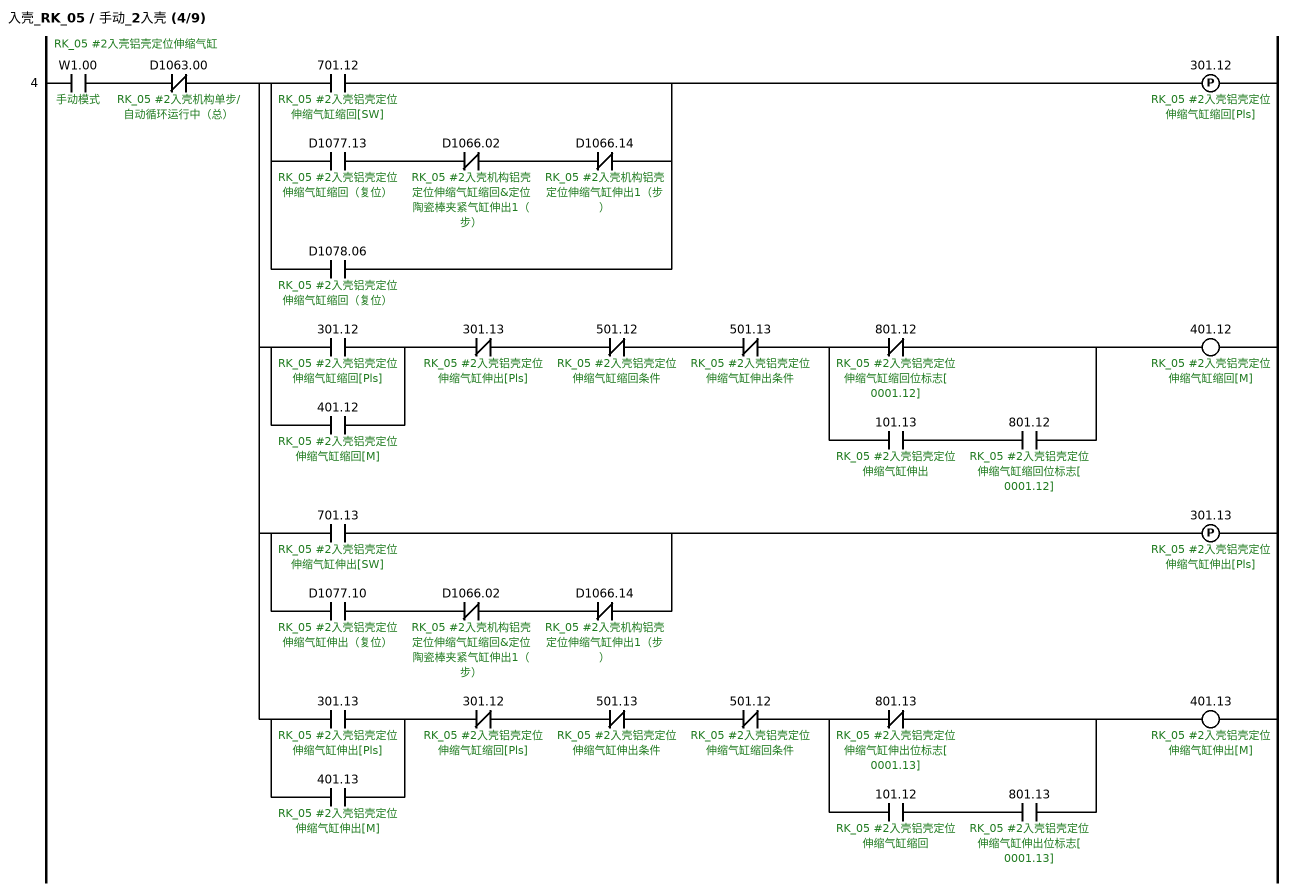
; [picture p432: 入壳_RK_05 / 手动_2入壳, rungs 4-4]
; rung 4: RK_05 #2入壳铝壳定位伸缩气缸
LD W1.00  ; 手动模式
ANDNOT D1063.00  ; RK_05 #2入壳机构单步/自动循环运行中（总）
OUT TR0
LD 701.12  ; RK_05 #2入壳铝壳定位伸缩气缸缩回[SW]
LD D1077.13  ; RK_05 #2入壳铝壳定位伸缩气缸缩回（复位）
ANDNOT D1066.02  ; RK_05 #2入壳机构铝壳定位伸缩气缸缩回&定位陶瓷棒夹紧气缸伸出1（步）
ANDNOT D1066.14  ; RK_05 #2入壳机构铝壳定位伸缩气缸伸出1（步）
ORLD
OR D1078.06  ; RK_05 #2入壳铝壳定位伸缩气缸缩回（复位）
ANDLD
DIFU(013) 301.12  ; RK_05 #2入壳铝壳定位伸缩气缸缩回[Pls]
LD TR0
LD 301.12  ; RK_05 #2入壳铝壳定位伸缩气缸缩回[Pls]
OR 401.12  ; RK_05 #2入壳铝壳定位伸缩气缸缩回[M]
ANDLD
ANDNOT 301.13  ; RK_05 #2入壳铝壳定位伸缩气缸伸出[Pls]
ANDNOT 501.12  ; RK_05 #2入壳铝壳定位伸缩气缸缩回条件
ANDNOT 501.13  ; RK_05 #2入壳铝壳定位伸缩气缸伸出条件
LDNOT 801.12  ; RK_05 #2入壳铝壳定位伸缩气缸缩回位标志[0001.12]
LD 101.13  ; RK_05 #2入壳铝壳定位伸缩气缸伸出
AND 801.12  ; RK_05 #2入壳铝壳定位伸缩气缸缩回位标志[0001.12]
ORLD
ANDLD
OUT 401.12  ; RK_05 #2入壳铝壳定位伸缩气缸缩回[M]
LD TR0
LD 701.13  ; RK_05 #2入壳铝壳定位伸缩气缸伸出[SW]
LD D1077.10  ; RK_05 #2入壳铝壳定位伸缩气缸伸出（复位）
ANDNOT D1066.02  ; RK_05 #2入壳机构铝壳定位伸缩气缸缩回&定位陶瓷棒夹紧气缸伸出1（步）
ANDNOT D1066.14  ; RK_05 #2入壳机构铝壳定位伸缩气缸伸出1（步）
ORLD
ANDLD
DIFU(013) 301.13  ; RK_05 #2入壳铝壳定位伸缩气缸伸出[Pls]
LD TR0
LD 301.13  ; RK_05 #2入壳铝壳定位伸缩气缸伸出[Pls]
OR 401.13  ; RK_05 #2入壳铝壳定位伸缩气缸伸出[M]
ANDLD
ANDNOT 301.12  ; RK_05 #2入壳铝壳定位伸缩气缸缩回[Pls]
ANDNOT 501.13  ; RK_05 #2入壳铝壳定位伸缩气缸伸出条件
ANDNOT 501.12  ; RK_05 #2入壳铝壳定位伸缩气缸缩回条件
LDNOT 801.13  ; RK_05 #2入壳铝壳定位伸缩气缸伸出位标志[0001.13]
LD 101.12  ; RK_05 #2入壳铝壳定位伸缩气缸缩回
AND 801.13  ; RK_05 #2入壳铝壳定位伸缩气缸伸出位标志[0001.13]
ORLD
ANDLD
OUT 401.13  ; RK_05 #2入壳铝壳定位伸缩气缸伸出[M]

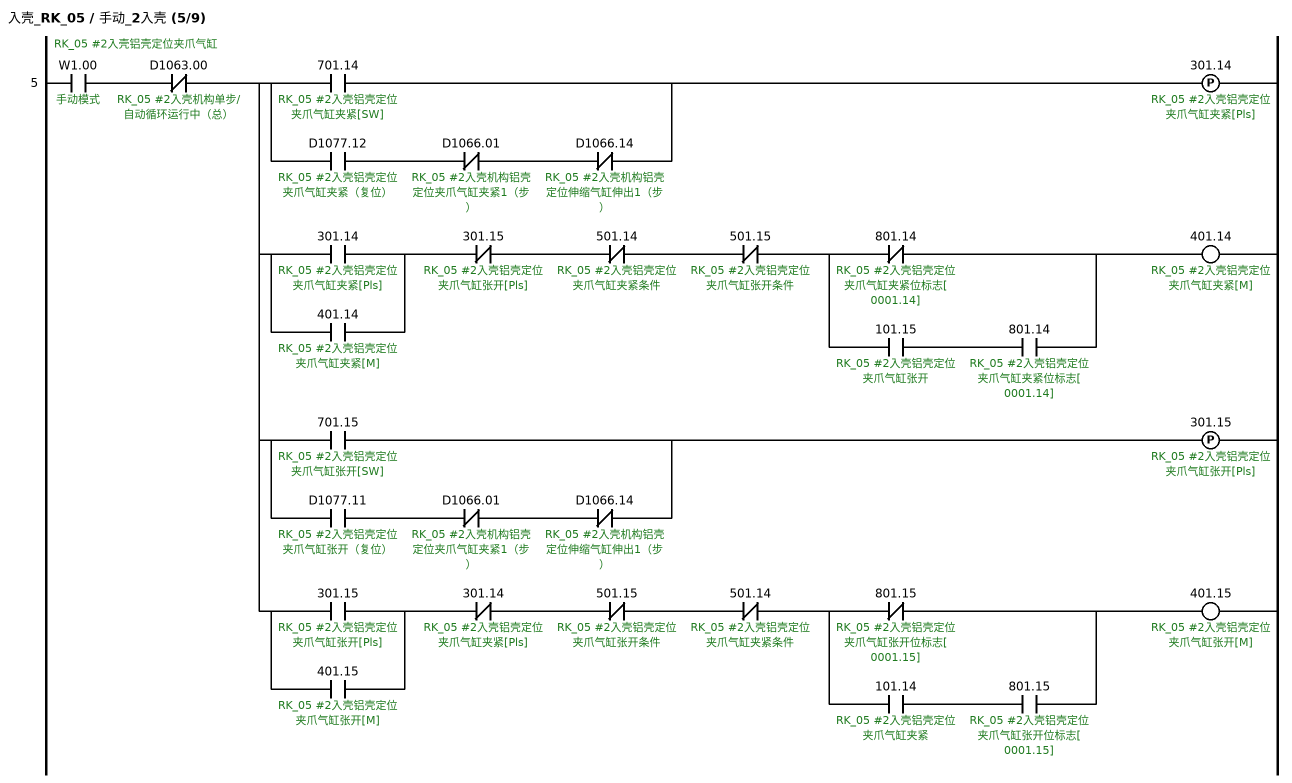
; rung 5: RK_05 #2入壳铝壳定位夹爪气缸
LD W1.00  ; 手动模式
ANDNOT D1063.00  ; RK_05 #2入壳机构单步/自动循环运行中（总）
OUT TR0
LD 701.14  ; RK_05 #2入壳铝壳定位夹爪气缸夹紧[SW]
LD D1077.12  ; RK_05 #2入壳铝壳定位夹爪气缸夹紧（复位）
ANDNOT D1066.01  ; RK_05 #2入壳机构铝壳定位夹爪气缸夹紧1（步）
ANDNOT D1066.14  ; RK_05 #2入壳机构铝壳定位伸缩气缸伸出1（步）
ORLD
ANDLD
DIFU(013) 301.14  ; RK_05 #2入壳铝壳定位夹爪气缸夹紧[Pls]
LD TR0
LD 301.14  ; RK_05 #2入壳铝壳定位夹爪气缸夹紧[Pls]
OR 401.14  ; RK_05 #2入壳铝壳定位夹爪气缸夹紧[M]
ANDLD
ANDNOT 301.15  ; RK_05 #2入壳铝壳定位夹爪气缸张开[Pls]
ANDNOT 501.14  ; RK_05 #2入壳铝壳定位夹爪气缸夹紧条件
ANDNOT 501.15  ; RK_05 #2入壳铝壳定位夹爪气缸张开条件
LDNOT 801.14  ; RK_05 #2入壳铝壳定位夹爪气缸夹紧位标志[0001.14]
LD 101.15  ; RK_05 #2入壳铝壳定位夹爪气缸张开
AND 801.14  ; RK_05 #2入壳铝壳定位夹爪气缸夹紧位标志[0001.14]
ORLD
ANDLD
OUT 401.14  ; RK_05 #2入壳铝壳定位夹爪气缸夹紧[M]
LD TR0
LD 701.15  ; RK_05 #2入壳铝壳定位夹爪气缸张开[SW]
LD D1077.11  ; RK_05 #2入壳铝壳定位夹爪气缸张开（复位）
ANDNOT D1066.01  ; RK_05 #2入壳机构铝壳定位夹爪气缸夹紧1（步）
ANDNOT D1066.14  ; RK_05 #2入壳机构铝壳定位伸缩气缸伸出1（步）
ORLD
ANDLD
DIFU(013) 301.15  ; RK_05 #2入壳铝壳定位夹爪气缸张开[Pls]
LD TR0
LD 301.15  ; RK_05 #2入壳铝壳定位夹爪气缸张开[Pls]
OR 401.15  ; RK_05 #2入壳铝壳定位夹爪气缸张开[M]
ANDLD
ANDNOT 301.14  ; RK_05 #2入壳铝壳定位夹爪气缸夹紧[Pls]
ANDNOT 501.15  ; RK_05 #2入壳铝壳定位夹爪气缸张开条件
ANDNOT 501.14  ; RK_05 #2入壳铝壳定位夹爪气缸夹紧条件
LDNOT 801.15  ; RK_05 #2入壳铝壳定位夹爪气缸张开位标志[0001.15]
LD 101.14  ; RK_05 #2入壳铝壳定位夹爪气缸夹紧
AND 801.15  ; RK_05 #2入壳铝壳定位夹爪气缸张开位标志[0001.15]
ORLD
ANDLD
OUT 401.15  ; RK_05 #2入壳铝壳定位夹爪气缸张开[M]

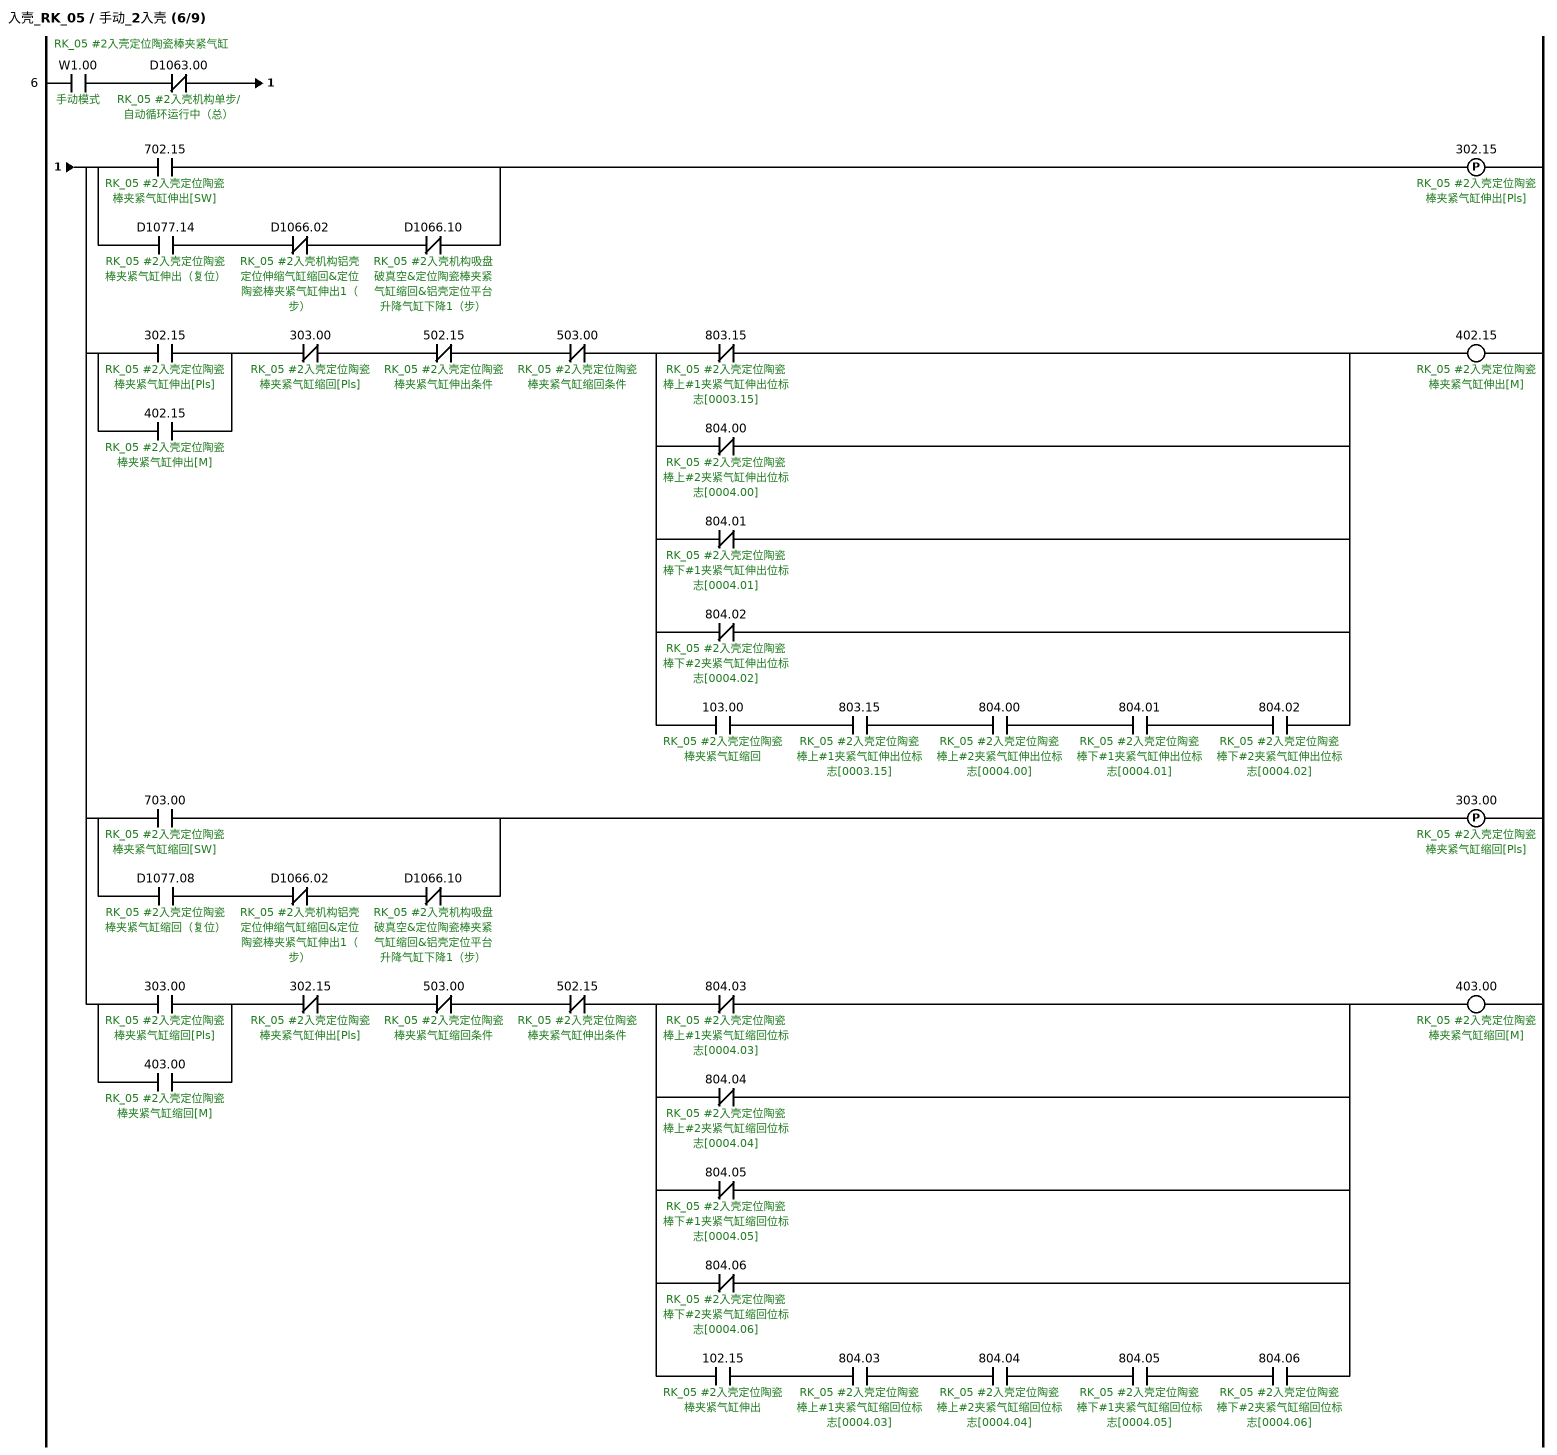
; rung 6: RK_05 #2入壳定位陶瓷棒夹紧气缸
LD W1.00  ; 手动模式
ANDNOT D1063.00  ; RK_05 #2入壳机构单步/自动循环运行中（总）
OUT TR0
LD 702.15  ; RK_05 #2入壳定位陶瓷棒夹紧气缸伸出[SW]
LD D1077.14  ; RK_05 #2入壳定位陶瓷棒夹紧气缸伸出（复位）
ANDNOT D1066.02  ; RK_05 #2入壳机构铝壳定位伸缩气缸缩回&定位陶瓷棒夹紧气缸伸出1（步）
ANDNOT D1066.10  ; RK_05 #2入壳机构吸盘破真空&定位陶瓷棒夹紧气缸缩回&铝壳定位平台升降气缸下降1（步）
ORLD
ANDLD
DIFU(013) 302.15  ; RK_05 #2入壳定位陶瓷棒夹紧气缸伸出[Pls]
LD TR0
LD 302.15  ; RK_05 #2入壳定位陶瓷棒夹紧气缸伸出[Pls]
OR 402.15  ; RK_05 #2入壳定位陶瓷棒夹紧气缸伸出[M]
ANDLD
ANDNOT 303.00  ; RK_05 #2入壳定位陶瓷棒夹紧气缸缩回[Pls]
ANDNOT 502.15  ; RK_05 #2入壳定位陶瓷棒夹紧气缸伸出条件
ANDNOT 503.00  ; RK_05 #2入壳定位陶瓷棒夹紧气缸缩回条件
LDNOT 803.15  ; RK_05 #2入壳定位陶瓷棒上#1夹紧气缸伸出位标志[0003.15]
ORNOT 804.00  ; RK_05 #2入壳定位陶瓷棒上#2夹紧气缸伸出位标志[0004.00]
ORNOT 804.01  ; RK_05 #2入壳定位陶瓷棒下#1夹紧气缸伸出位标志[0004.01]
ORNOT 804.02  ; RK_05 #2入壳定位陶瓷棒下#2夹紧气缸伸出位标志[0004.02]
LD 103.00  ; RK_05 #2入壳定位陶瓷棒夹紧气缸缩回
AND 803.15  ; RK_05 #2入壳定位陶瓷棒上#1夹紧气缸伸出位标志[0003.15]
AND 804.00  ; RK_05 #2入壳定位陶瓷棒上#2夹紧气缸伸出位标志[0004.00]
AND 804.01  ; RK_05 #2入壳定位陶瓷棒下#1夹紧气缸伸出位标志[0004.01]
AND 804.02  ; RK_05 #2入壳定位陶瓷棒下#2夹紧气缸伸出位标志[0004.02]
ORLD
ANDLD
OUT 402.15  ; RK_05 #2入壳定位陶瓷棒夹紧气缸伸出[M]
LD TR0
LD 703.00  ; RK_05 #2入壳定位陶瓷棒夹紧气缸缩回[SW]
LD D1077.08  ; RK_05 #2入壳定位陶瓷棒夹紧气缸缩回（复位）
ANDNOT D1066.02  ; RK_05 #2入壳机构铝壳定位伸缩气缸缩回&定位陶瓷棒夹紧气缸伸出1（步）
ANDNOT D1066.10  ; RK_05 #2入壳机构吸盘破真空&定位陶瓷棒夹紧气缸缩回&铝壳定位平台升降气缸下降1（步）
ORLD
ANDLD
DIFU(013) 303.00  ; RK_05 #2入壳定位陶瓷棒夹紧气缸缩回[Pls]
LD TR0
LD 303.00  ; RK_05 #2入壳定位陶瓷棒夹紧气缸缩回[Pls]
OR 403.00  ; RK_05 #2入壳定位陶瓷棒夹紧气缸缩回[M]
ANDLD
ANDNOT 302.15  ; RK_05 #2入壳定位陶瓷棒夹紧气缸伸出[Pls]
ANDNOT 503.00  ; RK_05 #2入壳定位陶瓷棒夹紧气缸缩回条件
ANDNOT 502.15  ; RK_05 #2入壳定位陶瓷棒夹紧气缸伸出条件
LDNOT 804.03  ; RK_05 #2入壳定位陶瓷棒上#1夹紧气缸缩回位标志[0004.03]
ORNOT 804.04  ; RK_05 #2入壳定位陶瓷棒上#2夹紧气缸缩回位标志[0004.04]
ORNOT 804.05  ; RK_05 #2入壳定位陶瓷棒下#1夹紧气缸缩回位标志[0004.05]
ORNOT 804.06  ; RK_05 #2入壳定位陶瓷棒下#2夹紧气缸缩回位标志[0004.06]
LD 102.15  ; RK_05 #2入壳定位陶瓷棒夹紧气缸伸出
AND 804.03  ; RK_05 #2入壳定位陶瓷棒上#1夹紧气缸缩回位标志[0004.03]
AND 804.04  ; RK_05 #2入壳定位陶瓷棒上#2夹紧气缸缩回位标志[0004.04]
AND 804.05  ; RK_05 #2入壳定位陶瓷棒下#1夹紧气缸缩回位标志[0004.05]
AND 804.06  ; RK_05 #2入壳定位陶瓷棒下#2夹紧气缸缩回位标志[0004.06]
ORLD
ANDLD
OUT 403.00  ; RK_05 #2入壳定位陶瓷棒夹紧气缸缩回[M]

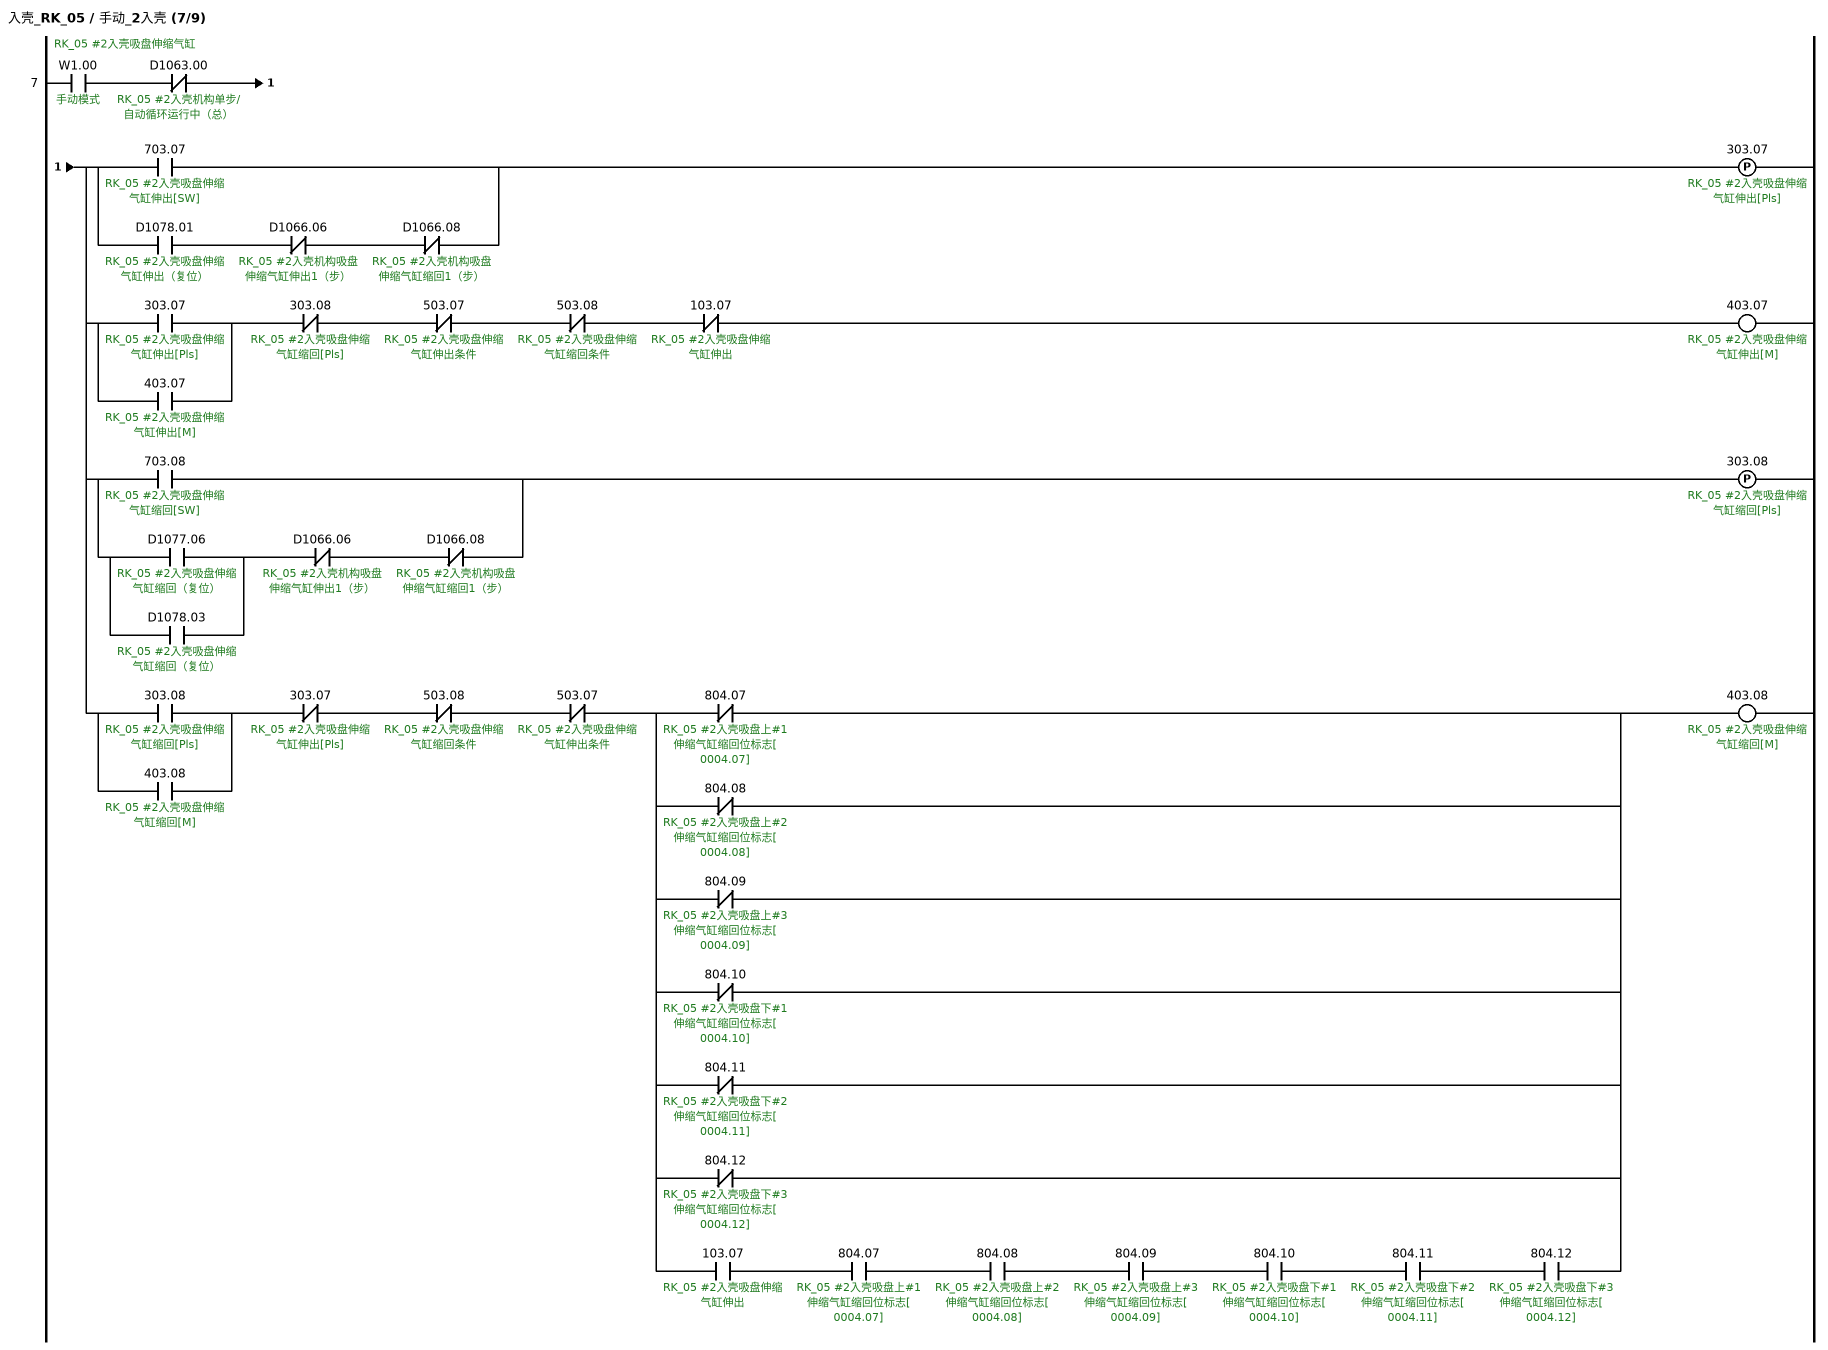
; rung 7: RK_05 #2入壳吸盘伸缩气缸
LD W1.00  ; 手动模式
ANDNOT D1063.00  ; RK_05 #2入壳机构单步/自动循环运行中（总）
OUT TR0
LD 703.07  ; RK_05 #2入壳吸盘伸缩气缸伸出[SW]
LD D1078.01  ; RK_05 #2入壳吸盘伸缩气缸伸出（复位）
ANDNOT D1066.06  ; RK_05 #2入壳机构吸盘伸缩气缸伸出1（步）
ANDNOT D1066.08  ; RK_05 #2入壳机构吸盘伸缩气缸缩回1（步）
ORLD
ANDLD
DIFU(013) 303.07  ; RK_05 #2入壳吸盘伸缩气缸伸出[Pls]
LD TR0
LD 303.07  ; RK_05 #2入壳吸盘伸缩气缸伸出[Pls]
OR 403.07  ; RK_05 #2入壳吸盘伸缩气缸伸出[M]
ANDLD
ANDNOT 303.08  ; RK_05 #2入壳吸盘伸缩气缸缩回[Pls]
ANDNOT 503.07  ; RK_05 #2入壳吸盘伸缩气缸伸出条件
ANDNOT 503.08  ; RK_05 #2入壳吸盘伸缩气缸缩回条件
ANDNOT 103.07  ; RK_05 #2入壳吸盘伸缩气缸伸出
OUT 403.07  ; RK_05 #2入壳吸盘伸缩气缸伸出[M]
LD TR0
LD 703.08  ; RK_05 #2入壳吸盘伸缩气缸缩回[SW]
LD D1077.06  ; RK_05 #2入壳吸盘伸缩气缸缩回（复位）
OR D1078.03  ; RK_05 #2入壳吸盘伸缩气缸缩回（复位）
ANDNOT D1066.06  ; RK_05 #2入壳机构吸盘伸缩气缸伸出1（步）
ANDNOT D1066.08  ; RK_05 #2入壳机构吸盘伸缩气缸缩回1（步）
ORLD
ANDLD
DIFU(013) 303.08  ; RK_05 #2入壳吸盘伸缩气缸缩回[Pls]
LD TR0
LD 303.08  ; RK_05 #2入壳吸盘伸缩气缸缩回[Pls]
OR 403.08  ; RK_05 #2入壳吸盘伸缩气缸缩回[M]
ANDLD
ANDNOT 303.07  ; RK_05 #2入壳吸盘伸缩气缸伸出[Pls]
ANDNOT 503.08  ; RK_05 #2入壳吸盘伸缩气缸缩回条件
ANDNOT 503.07  ; RK_05 #2入壳吸盘伸缩气缸伸出条件
LDNOT 804.07  ; RK_05 #2入壳吸盘上#1伸缩气缸缩回位标志[0004.07]
ORNOT 804.08  ; RK_05 #2入壳吸盘上#2伸缩气缸缩回位标志[0004.08]
ORNOT 804.09  ; RK_05 #2入壳吸盘上#3伸缩气缸缩回位标志[0004.09]
ORNOT 804.10  ; RK_05 #2入壳吸盘下#1伸缩气缸缩回位标志[0004.10]
ORNOT 804.11  ; RK_05 #2入壳吸盘下#2伸缩气缸缩回位标志[0004.11]
ORNOT 804.12  ; RK_05 #2入壳吸盘下#3伸缩气缸缩回位标志[0004.12]
LD 103.07  ; RK_05 #2入壳吸盘伸缩气缸伸出
AND 804.07  ; RK_05 #2入壳吸盘上#1伸缩气缸缩回位标志[0004.07]
AND 804.08  ; RK_05 #2入壳吸盘上#2伸缩气缸缩回位标志[0004.08]
AND 804.09  ; RK_05 #2入壳吸盘上#3伸缩气缸缩回位标志[0004.09]
AND 804.10  ; RK_05 #2入壳吸盘下#1伸缩气缸缩回位标志[0004.10]
AND 804.11  ; RK_05 #2入壳吸盘下#2伸缩气缸缩回位标志[0004.11]
AND 804.12  ; RK_05 #2入壳吸盘下#3伸缩气缸缩回位标志[0004.12]
ORLD
ANDLD
OUT 403.08  ; RK_05 #2入壳吸盘伸缩气缸缩回[M]

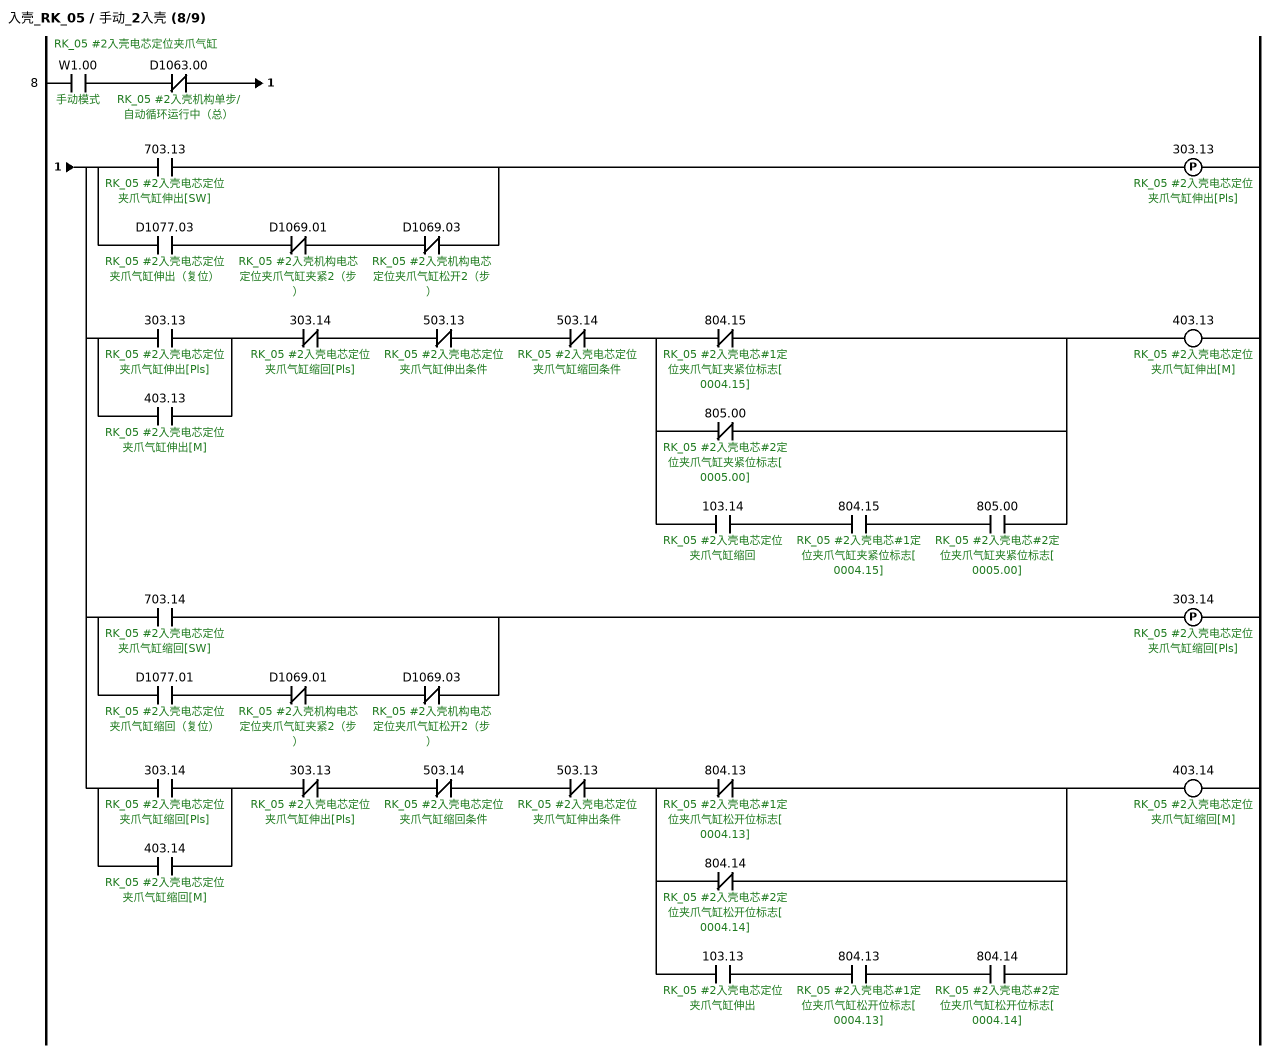
; rung 8: RK_05 #2入壳电芯定位夹爪气缸
LD W1.00  ; 手动模式
ANDNOT D1063.00  ; RK_05 #2入壳机构单步/自动循环运行中（总）
OUT TR0
LD 703.13  ; RK_05 #2入壳电芯定位夹爪气缸伸出[SW]
LD D1077.03  ; RK_05 #2入壳电芯定位夹爪气缸伸出（复位）
ANDNOT D1069.01  ; RK_05 #2入壳机构电芯定位夹爪气缸夹紧2（步）
ANDNOT D1069.03  ; RK_05 #2入壳机构电芯定位夹爪气缸松开2（步）
ORLD
ANDLD
DIFU(013) 303.13  ; RK_05 #2入壳电芯定位夹爪气缸伸出[Pls]
LD TR0
LD 303.13  ; RK_05 #2入壳电芯定位夹爪气缸伸出[Pls]
OR 403.13  ; RK_05 #2入壳电芯定位夹爪气缸伸出[M]
ANDLD
ANDNOT 303.14  ; RK_05 #2入壳电芯定位夹爪气缸缩回[Pls]
ANDNOT 503.13  ; RK_05 #2入壳电芯定位夹爪气缸伸出条件
ANDNOT 503.14  ; RK_05 #2入壳电芯定位夹爪气缸缩回条件
LDNOT 804.15  ; RK_05 #2入壳电芯#1定位夹爪气缸夹紧位标志[0004.15]
ORNOT 805.00  ; RK_05 #2入壳电芯#2定位夹爪气缸夹紧位标志[0005.00]
LD 103.14  ; RK_05 #2入壳电芯定位夹爪气缸缩回
AND 804.15  ; RK_05 #2入壳电芯#1定位夹爪气缸夹紧位标志[0004.15]
AND 805.00  ; RK_05 #2入壳电芯#2定位夹爪气缸夹紧位标志[0005.00]
ORLD
ANDLD
OUT 403.13  ; RK_05 #2入壳电芯定位夹爪气缸伸出[M]
LD TR0
LD 703.14  ; RK_05 #2入壳电芯定位夹爪气缸缩回[SW]
LD D1077.01  ; RK_05 #2入壳电芯定位夹爪气缸缩回（复位）
ANDNOT D1069.01  ; RK_05 #2入壳机构电芯定位夹爪气缸夹紧2（步）
ANDNOT D1069.03  ; RK_05 #2入壳机构电芯定位夹爪气缸松开2（步）
ORLD
ANDLD
DIFU(013) 303.14  ; RK_05 #2入壳电芯定位夹爪气缸缩回[Pls]
LD TR0
LD 303.14  ; RK_05 #2入壳电芯定位夹爪气缸缩回[Pls]
OR 403.14  ; RK_05 #2入壳电芯定位夹爪气缸缩回[M]
ANDLD
ANDNOT 303.13  ; RK_05 #2入壳电芯定位夹爪气缸伸出[Pls]
ANDNOT 503.14  ; RK_05 #2入壳电芯定位夹爪气缸缩回条件
ANDNOT 503.13  ; RK_05 #2入壳电芯定位夹爪气缸伸出条件
LDNOT 804.13  ; RK_05 #2入壳电芯#1定位夹爪气缸松开位标志[0004.13]
ORNOT 804.14  ; RK_05 #2入壳电芯#2定位夹爪气缸松开位标志[0004.14]
LD 103.13  ; RK_05 #2入壳电芯定位夹爪气缸伸出
AND 804.13  ; RK_05 #2入壳电芯#1定位夹爪气缸松开位标志[0004.13]
AND 804.14  ; RK_05 #2入壳电芯#2定位夹爪气缸松开位标志[0004.14]
ORLD
ANDLD
OUT 403.14  ; RK_05 #2入壳电芯定位夹爪气缸缩回[M]

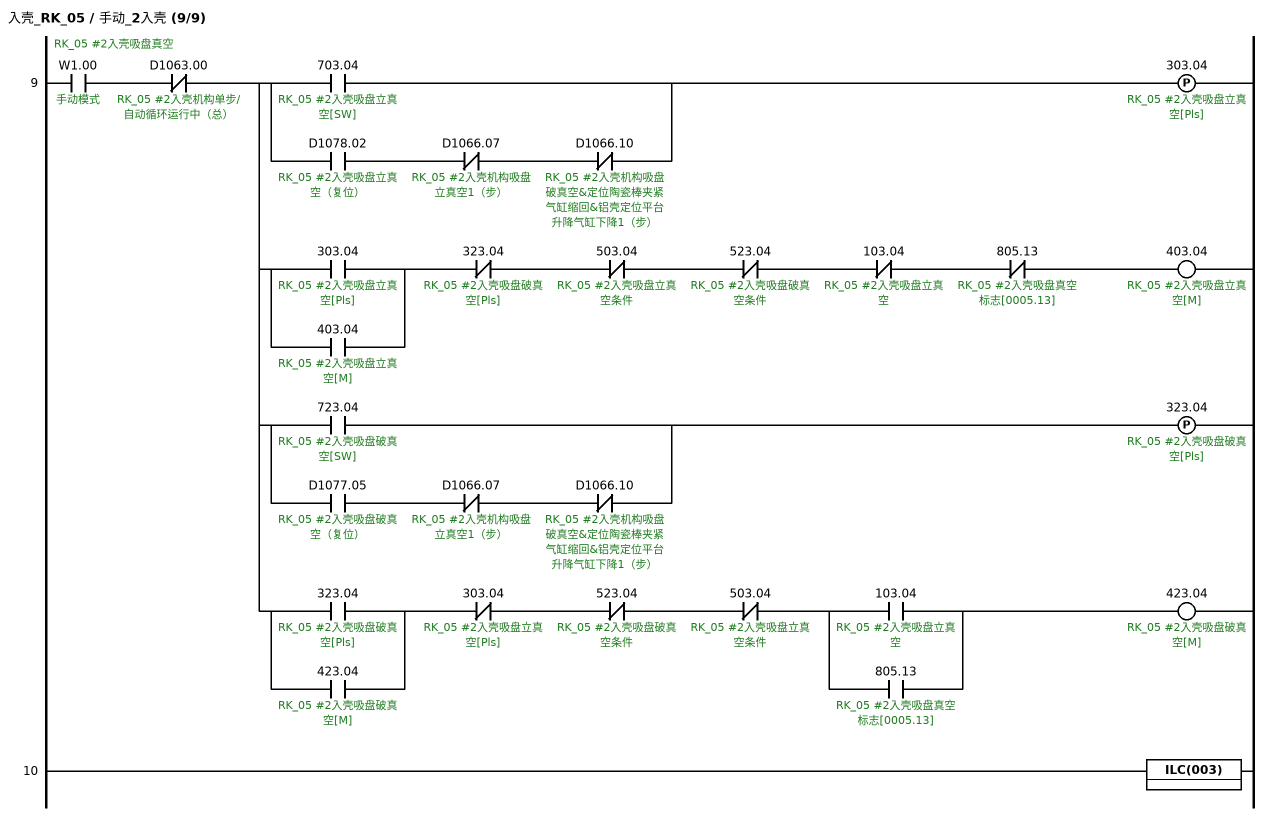
; rung 9: RK_05 #2入壳吸盘真空
LD W1.00  ; 手动模式
ANDNOT D1063.00  ; RK_05 #2入壳机构单步/自动循环运行中（总）
OUT TR0
LD 703.04  ; RK_05 #2入壳吸盘立真空[SW]
LD D1078.02  ; RK_05 #2入壳吸盘立真空（复位）
ANDNOT D1066.07  ; RK_05 #2入壳机构吸盘立真空1（步）
ANDNOT D1066.10  ; RK_05 #2入壳机构吸盘破真空&定位陶瓷棒夹紧气缸缩回&铝壳定位平台升降气缸下降1（步）
ORLD
ANDLD
DIFU(013) 303.04  ; RK_05 #2入壳吸盘立真空[Pls]
LD TR0
LD 303.04  ; RK_05 #2入壳吸盘立真空[Pls]
OR 403.04  ; RK_05 #2入壳吸盘立真空[M]
ANDLD
ANDNOT 323.04  ; RK_05 #2入壳吸盘破真空[Pls]
ANDNOT 503.04  ; RK_05 #2入壳吸盘立真空条件
ANDNOT 523.04  ; RK_05 #2入壳吸盘破真空条件
ANDNOT 103.04  ; RK_05 #2入壳吸盘立真空
ANDNOT 805.13  ; RK_05 #2入壳吸盘真空标志[0005.13]
OUT 403.04  ; RK_05 #2入壳吸盘立真空[M]
LD TR0
LD 723.04  ; RK_05 #2入壳吸盘破真空[SW]
LD D1077.05  ; RK_05 #2入壳吸盘破真空（复位）
ANDNOT D1066.07  ; RK_05 #2入壳机构吸盘立真空1（步）
ANDNOT D1066.10  ; RK_05 #2入壳机构吸盘破真空&定位陶瓷棒夹紧气缸缩回&铝壳定位平台升降气缸下降1（步）
ORLD
ANDLD
DIFU(013) 323.04  ; RK_05 #2入壳吸盘破真空[Pls]
LD TR0
LD 323.04  ; RK_05 #2入壳吸盘破真空[Pls]
OR 423.04  ; RK_05 #2入壳吸盘破真空[M]
ANDLD
ANDNOT 303.04  ; RK_05 #2入壳吸盘立真空[Pls]
ANDNOT 523.04  ; RK_05 #2入壳吸盘破真空条件
ANDNOT 503.04  ; RK_05 #2入壳吸盘立真空条件
LD 103.04  ; RK_05 #2入壳吸盘立真空
OR 805.13  ; RK_05 #2入壳吸盘真空标志[0005.13]
ANDLD
OUT 423.04  ; RK_05 #2入壳吸盘破真空[M]
; rung 10
ILC(003)

### Section 自动_1入壳

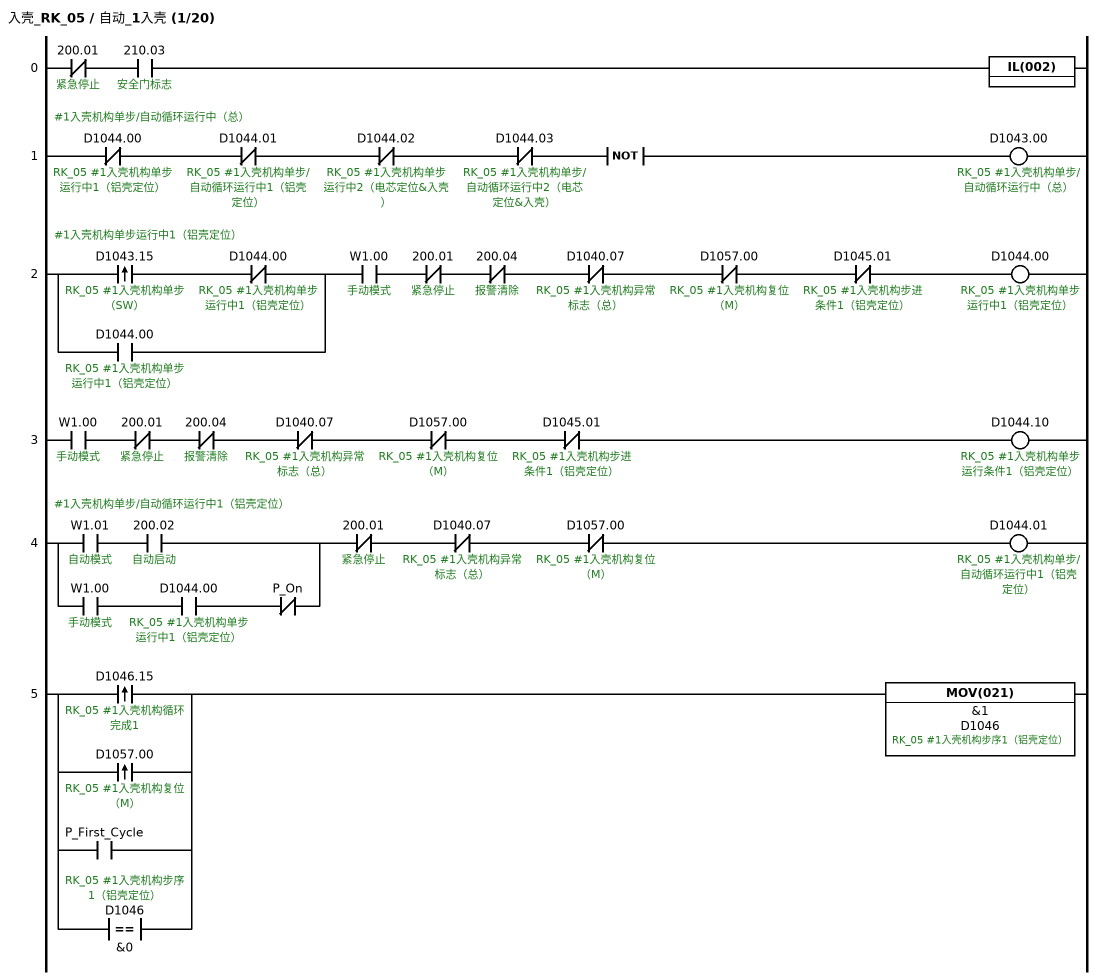
; rung 0
LDNOT 200.01  ; 紧急停止
AND 210.03  ; 安全门标志
IL(002)
; rung 1: #1入壳机构单步/自动循环运行中（总）
LDNOT D1044.00  ; RK_05 #1入壳机构单步运行中1（铝壳定位）
ANDNOT D1044.01  ; RK_05 #1入壳机构单步/自动循环运行中1（铝壳定位）
ANDNOT D1044.02  ; RK_05 #1入壳机构单步运行中2（电芯定位&入壳）
ANDNOT D1044.03  ; RK_05 #1入壳机构单步/自动循环运行中2（电芯定位&入壳）
NOT(520)
OUT D1043.00  ; RK_05 #1入壳机构单步/自动循环运行中（总）
; rung 2: #1入壳机构单步运行中1（铝壳定位）
@LD D1043.15  ; RK_05 #1入壳机构单步（SW）
ANDNOT D1044.00  ; RK_05 #1入壳机构单步运行中1（铝壳定位）
OR D1044.00  ; RK_05 #1入壳机构单步运行中1（铝壳定位）
AND W1.00  ; 手动模式
ANDNOT 200.01  ; 紧急停止
ANDNOT 200.04  ; 报警清除
ANDNOT D1040.07  ; RK_05 #1入壳机构异常标志（总）
ANDNOT D1057.00  ; RK_05 #1入壳机构复位（M）
ANDNOT D1045.01  ; RK_05 #1入壳机构步进条件1（铝壳定位）
OUT D1044.00  ; RK_05 #1入壳机构单步运行中1（铝壳定位）
; rung 3
LD W1.00  ; 手动模式
ANDNOT 200.01  ; 紧急停止
ANDNOT 200.04  ; 报警清除
ANDNOT D1040.07  ; RK_05 #1入壳机构异常标志（总）
ANDNOT D1057.00  ; RK_05 #1入壳机构复位（M）
ANDNOT D1045.01  ; RK_05 #1入壳机构步进条件1（铝壳定位）
OUT D1044.10  ; RK_05 #1入壳机构单步运行条件1（铝壳定位）
; rung 4: #1入壳机构单步/自动循环运行中1（铝壳定位）
LD W1.01  ; 自动模式
AND 200.02  ; 自动启动
LD W1.00  ; 手动模式
AND D1044.00  ; RK_05 #1入壳机构单步运行中1（铝壳定位）
ANDNOT P_On
ORLD
ANDNOT 200.01  ; 紧急停止
ANDNOT D1040.07  ; RK_05 #1入壳机构异常标志（总）
ANDNOT D1057.00  ; RK_05 #1入壳机构复位（M）
OUT D1044.01  ; RK_05 #1入壳机构单步/自动循环运行中1（铝壳定位）
; rung 5
@LD D1046.15  ; RK_05 #1入壳机构循环完成1
@OR D1057.00  ; RK_05 #1入壳机构复位（M）
OR P_First_Cycle
OR=(300) D1046 &0  ; RK_05 #1入壳机构步序1（铝壳定位）
MOV(021) &1 D1046  ; RK_05 #1入壳机构步序1（铝壳定位）

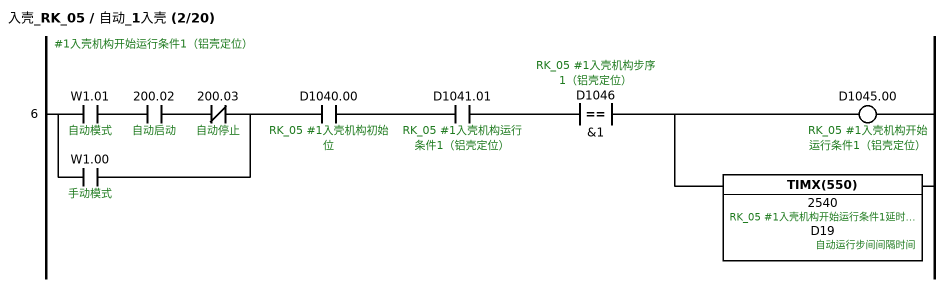
; rung 6: #1入壳机构开始运行条件1（铝壳定位）
LD W1.01  ; 自动模式
AND 200.02  ; 自动启动
ANDNOT 200.03  ; 自动停止
OR W1.00  ; 手动模式
AND D1040.00  ; RK_05 #1入壳机构初始位
AND D1041.01  ; RK_05 #1入壳机构运行条件1（铝壳定位）
AND=(300) D1046 &1  ; RK_05 #1入壳机构步序1（铝壳定位）
OUT D1045.00  ; RK_05 #1入壳机构开始运行条件1（铝壳定位）
TIMX(550) 2540 D19  ; 自动运行步间间隔时间, RK_05 #1入壳机构开始运行条件1延时（铝壳定位）

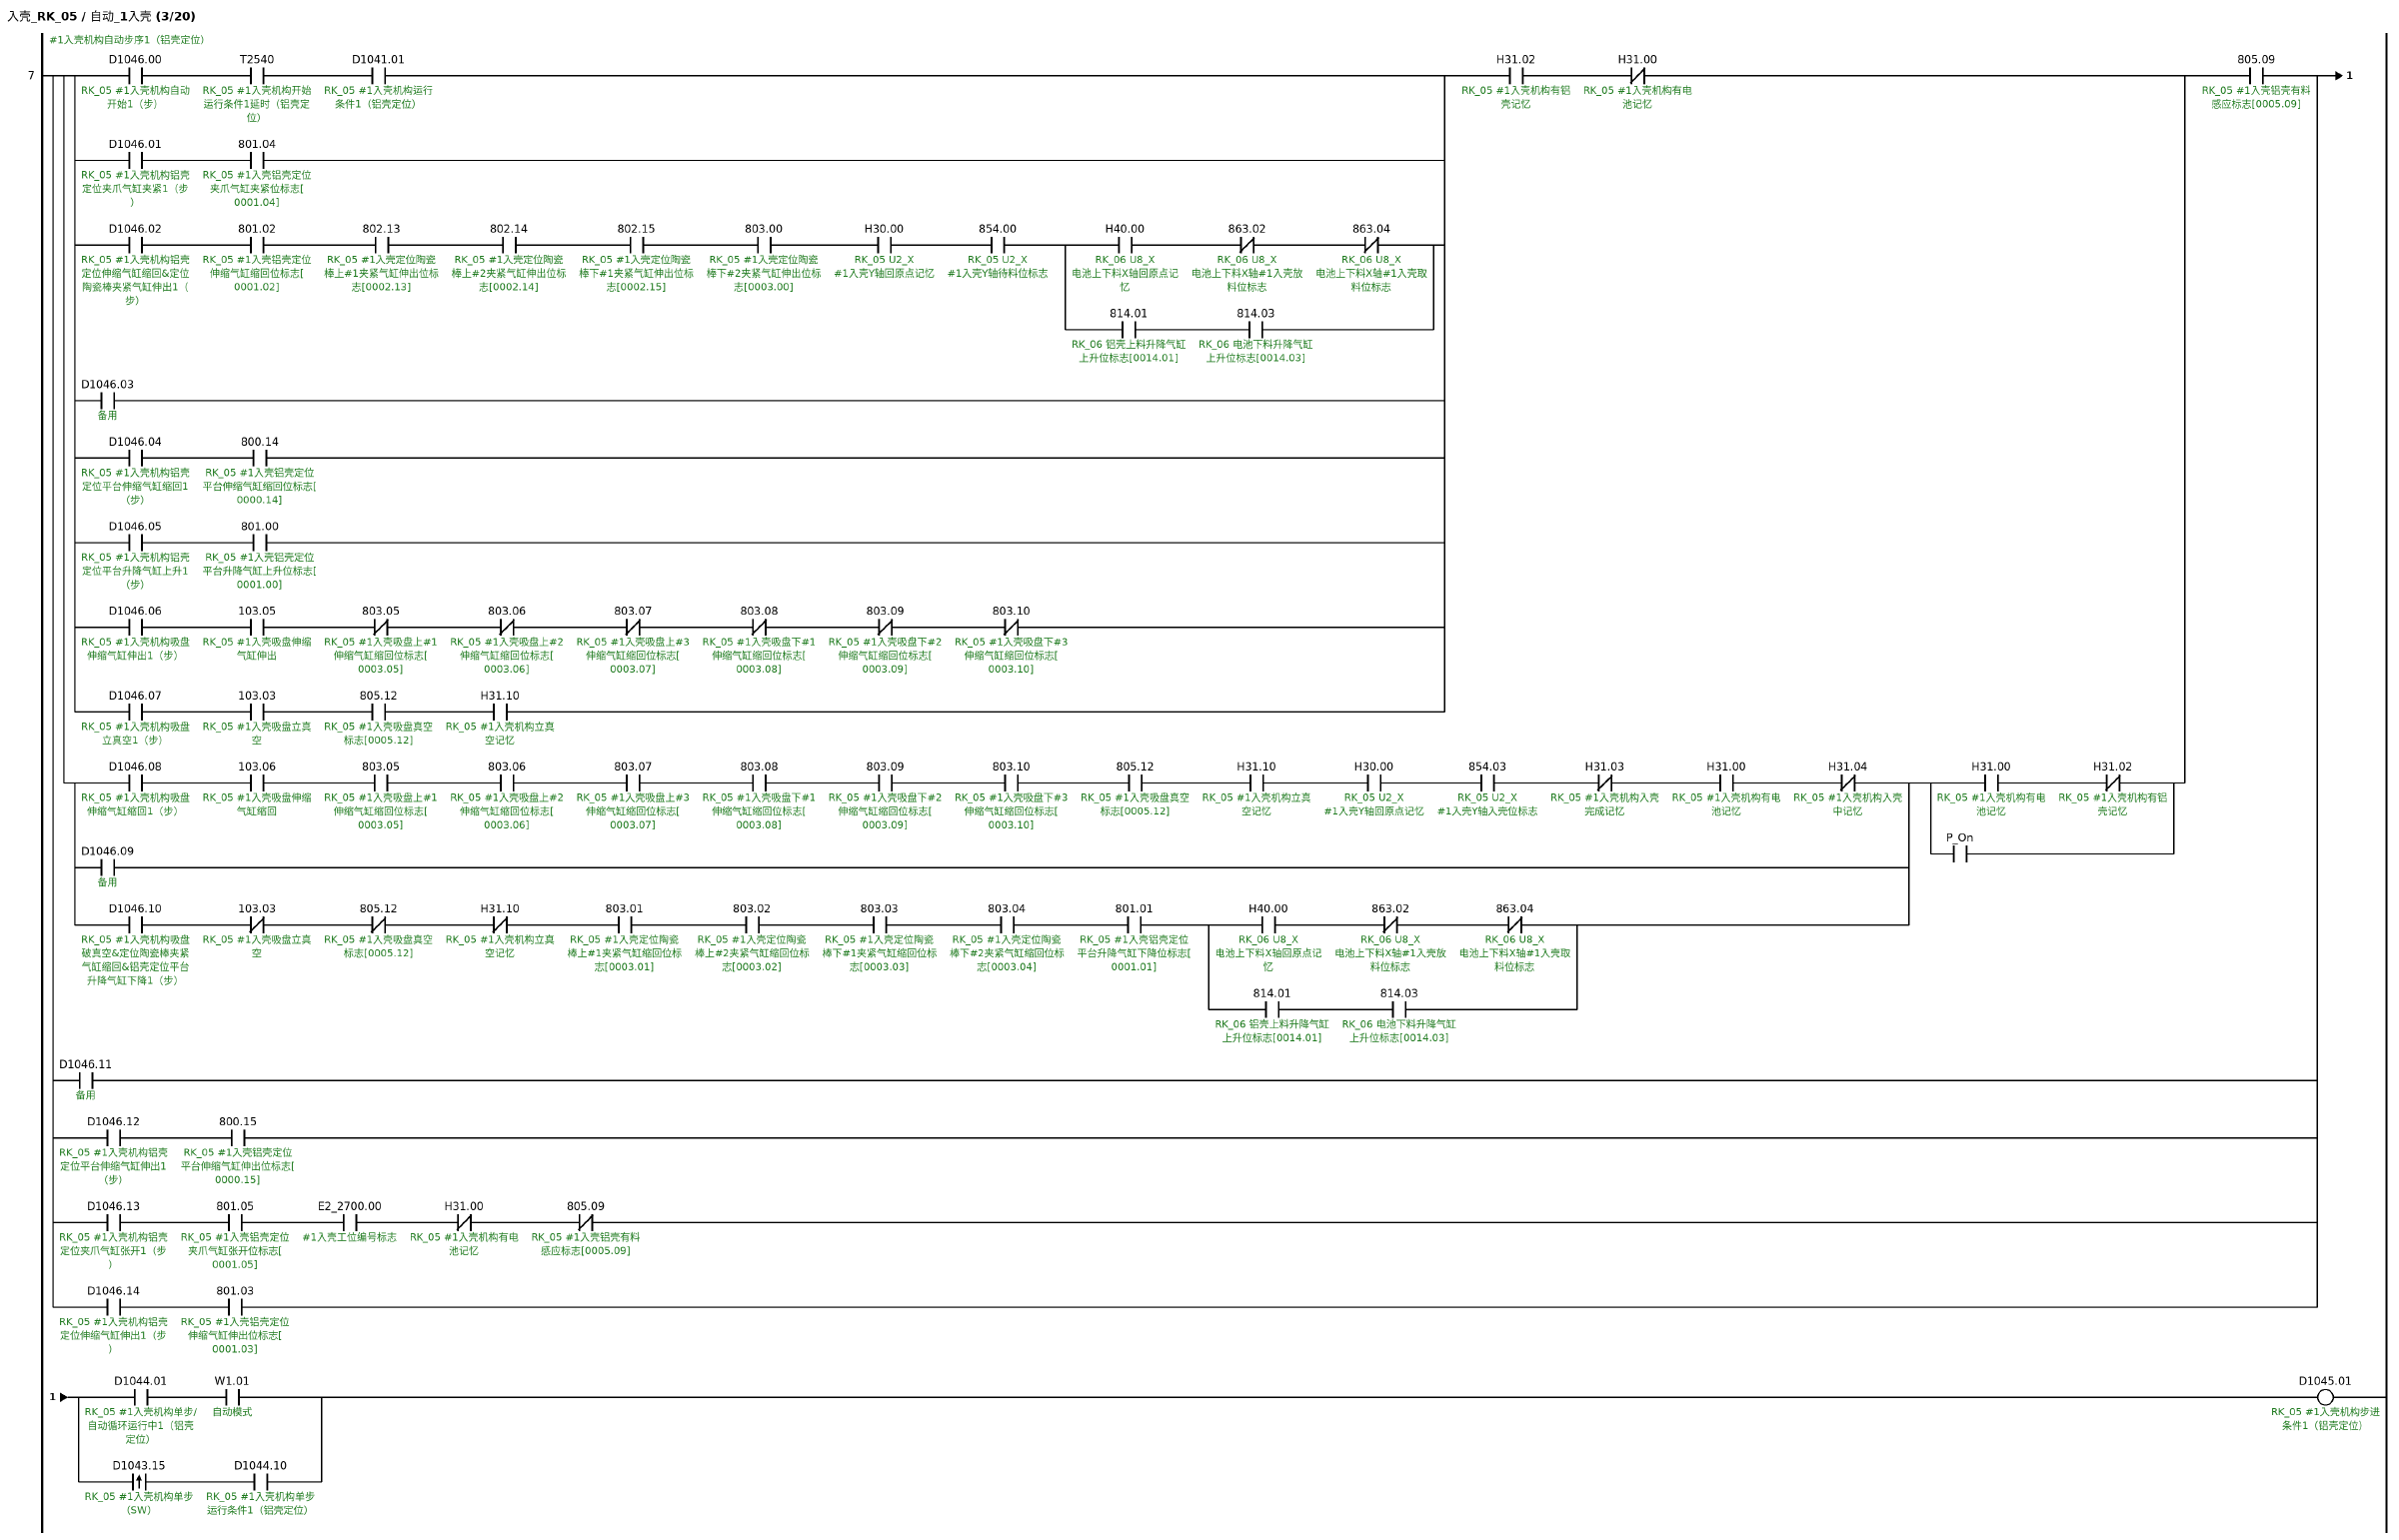
; rung 7: #1入壳机构自动步序1（铝壳定位）
LD D1046.00  ; RK_05 #1入壳机构自动开始1（步）
AND T2540  ; RK_05 #1入壳机构开始运行条件1延时（铝壳定位）
AND D1041.01  ; RK_05 #1入壳机构运行条件1（铝壳定位）
LD D1046.01  ; RK_05 #1入壳机构铝壳定位夹爪气缸夹紧1（步）
AND 801.04  ; RK_05 #1入壳铝壳定位夹爪气缸夹紧位标志[0001.04]
ORLD
LD D1046.02  ; RK_05 #1入壳机构铝壳定位伸缩气缸缩回&定位陶瓷棒夹紧气缸伸出1（步）
AND 801.02  ; RK_05 #1入壳铝壳定位伸缩气缸缩回位标志[0001.02]
AND 802.13  ; RK_05 #1入壳定位陶瓷棒上#1夹紧气缸伸出位标志[0002.13]
AND 802.14  ; RK_05 #1入壳定位陶瓷棒上#2夹紧气缸伸出位标志[0002.14]
AND 802.15  ; RK_05 #1入壳定位陶瓷棒下#1夹紧气缸伸出位标志[0002.15]
AND 803.00  ; RK_05 #1入壳定位陶瓷棒下#2夹紧气缸伸出位标志[0003.00]
AND H30.00  ; RK_05 U2_X #1入壳Y轴回原点记忆
AND 854.00  ; RK_05 U2_X #1入壳Y轴待料位标志
LD H40.00  ; RK_06 U8_X 电池上下料X轴回原点记忆
ANDNOT 863.02  ; RK_06 U8_X 电池上下料X轴#1入壳放料位标志
ANDNOT 863.04  ; RK_06 U8_X 电池上下料X轴#1入壳取料位标志
LD 814.01  ; RK_06 铝壳上料升降气缸上升位标志[0014.01]
AND 814.03  ; RK_06 电池下料升降气缸上升位标志[0014.03]
ORLD
ANDLD
ORLD
OR D1046.03  ; 备用
LD D1046.04  ; RK_05 #1入壳机构铝壳定位平台伸缩气缸缩回1（步）
AND 800.14  ; RK_05 #1入壳铝壳定位平台伸缩气缸缩回位标志[0000.14]
ORLD
LD D1046.05  ; RK_05 #1入壳机构铝壳定位平台升降气缸上升1（步）
AND 801.00  ; RK_05 #1入壳铝壳定位平台升降气缸上升位标志[0001.00]
ORLD
LD D1046.06  ; RK_05 #1入壳机构吸盘伸缩气缸伸出1（步）
AND 103.05  ; RK_05 #1入壳吸盘伸缩气缸伸出
ANDNOT 803.05  ; RK_05 #1入壳吸盘上#1伸缩气缸缩回位标志[0003.05]
ANDNOT 803.06  ; RK_05 #1入壳吸盘上#2伸缩气缸缩回位标志[0003.06]
ANDNOT 803.07  ; RK_05 #1入壳吸盘上#3伸缩气缸缩回位标志[0003.07]
ANDNOT 803.08  ; RK_05 #1入壳吸盘下#1伸缩气缸缩回位标志[0003.08]
ANDNOT 803.09  ; RK_05 #1入壳吸盘下#2伸缩气缸缩回位标志[0003.09]
ANDNOT 803.10  ; RK_05 #1入壳吸盘下#3伸缩气缸缩回位标志[0003.10]
ORLD
LD D1046.07  ; RK_05 #1入壳机构吸盘立真空1（步）
AND 103.03  ; RK_05 #1入壳吸盘立真空
AND 805.12  ; RK_05 #1入壳吸盘真空标志[0005.12]
AND H31.10  ; RK_05 #1入壳机构立真空记忆
ORLD
AND H31.02  ; RK_05 #1入壳机构有铝壳记忆
ANDNOT H31.00  ; RK_05 #1入壳机构有电池记忆
LD D1046.08  ; RK_05 #1入壳机构吸盘伸缩气缸缩回1（步）
AND 103.06  ; RK_05 #1入壳吸盘伸缩气缸缩回
AND 803.05  ; RK_05 #1入壳吸盘上#1伸缩气缸缩回位标志[0003.05]
AND 803.06  ; RK_05 #1入壳吸盘上#2伸缩气缸缩回位标志[0003.06]
AND 803.07  ; RK_05 #1入壳吸盘上#3伸缩气缸缩回位标志[0003.07]
AND 803.08  ; RK_05 #1入壳吸盘下#1伸缩气缸缩回位标志[0003.08]
AND 803.09  ; RK_05 #1入壳吸盘下#2伸缩气缸缩回位标志[0003.09]
AND 803.10  ; RK_05 #1入壳吸盘下#3伸缩气缸缩回位标志[0003.10]
AND 805.12  ; RK_05 #1入壳吸盘真空标志[0005.12]
AND H31.10  ; RK_05 #1入壳机构立真空记忆
AND H30.00  ; RK_05 U2_X #1入壳Y轴回原点记忆
AND 854.03  ; RK_05 U2_X #1入壳Y轴入壳位标志
ANDNOT H31.03  ; RK_05 #1入壳机构入壳完成记忆
AND H31.00  ; RK_05 #1入壳机构有电池记忆
ANDNOT H31.04  ; RK_05 #1入壳机构入壳中记忆
OR D1046.09  ; 备用
LD D1046.10  ; RK_05 #1入壳机构吸盘破真空&定位陶瓷棒夹紧气缸缩回&铝壳定位平台升降气缸下降1（步）
ANDNOT 103.03  ; RK_05 #1入壳吸盘立真空
ANDNOT 805.12  ; RK_05 #1入壳吸盘真空标志[0005.12]
ANDNOT H31.10  ; RK_05 #1入壳机构立真空记忆
AND 803.01  ; RK_05 #1入壳定位陶瓷棒上#1夹紧气缸缩回位标志[0003.01]
AND 803.02  ; RK_05 #1入壳定位陶瓷棒上#2夹紧气缸缩回位标志[0003.02]
AND 803.03  ; RK_05 #1入壳定位陶瓷棒下#1夹紧气缸缩回位标志[0003.03]
AND 803.04  ; RK_05 #1入壳定位陶瓷棒下#2夹紧气缸缩回位标志[0003.04]
AND 801.01  ; RK_05 #1入壳铝壳定位平台升降气缸下降位标志[0001.01]
LD H40.00  ; RK_06 U8_X 电池上下料X轴回原点记忆
ANDNOT 863.02  ; RK_06 U8_X 电池上下料X轴#1入壳放料位标志
ANDNOT 863.04  ; RK_06 U8_X 电池上下料X轴#1入壳取料位标志
LD 814.01  ; RK_06 铝壳上料升降气缸上升位标志[0014.01]
AND 814.03  ; RK_06 电池下料升降气缸上升位标志[0014.03]
ORLD
ANDLD
ORLD
LD H31.00  ; RK_05 #1入壳机构有电池记忆
ANDNOT H31.02  ; RK_05 #1入壳机构有铝壳记忆
OR P_On
ANDLD
ORLD
AND 805.09  ; RK_05 #1入壳铝壳有料感应标志[0005.09]
OR D1046.11  ; 备用
LD D1046.12  ; RK_05 #1入壳机构铝壳定位平台伸缩气缸伸出1（步）
AND 800.15  ; RK_05 #1入壳铝壳定位平台伸缩气缸伸出位标志[0000.15]
ORLD
LD D1046.13  ; RK_05 #1入壳机构铝壳定位夹爪气缸张开1（步）
AND 801.05  ; RK_05 #1入壳铝壳定位夹爪气缸张开位标志[0001.05]
AND E2_2700.00  ; #1入壳工位编号标志
ANDNOT H31.00  ; RK_05 #1入壳机构有电池记忆
ANDNOT 805.09  ; RK_05 #1入壳铝壳有料感应标志[0005.09]
ORLD
LD D1046.14  ; RK_05 #1入壳机构铝壳定位伸缩气缸伸出1（步）
AND 801.03  ; RK_05 #1入壳铝壳定位伸缩气缸伸出位标志[0001.03]
ORLD
LD D1044.01  ; RK_05 #1入壳机构单步/自动循环运行中1（铝壳定位）
AND W1.01  ; 自动模式
@LD D1043.15  ; RK_05 #1入壳机构单步（SW）
AND D1044.10  ; RK_05 #1入壳机构单步运行条件1（铝壳定位）
ORLD
ANDLD
OUT D1045.01  ; RK_05 #1入壳机构步进条件1（铝壳定位）

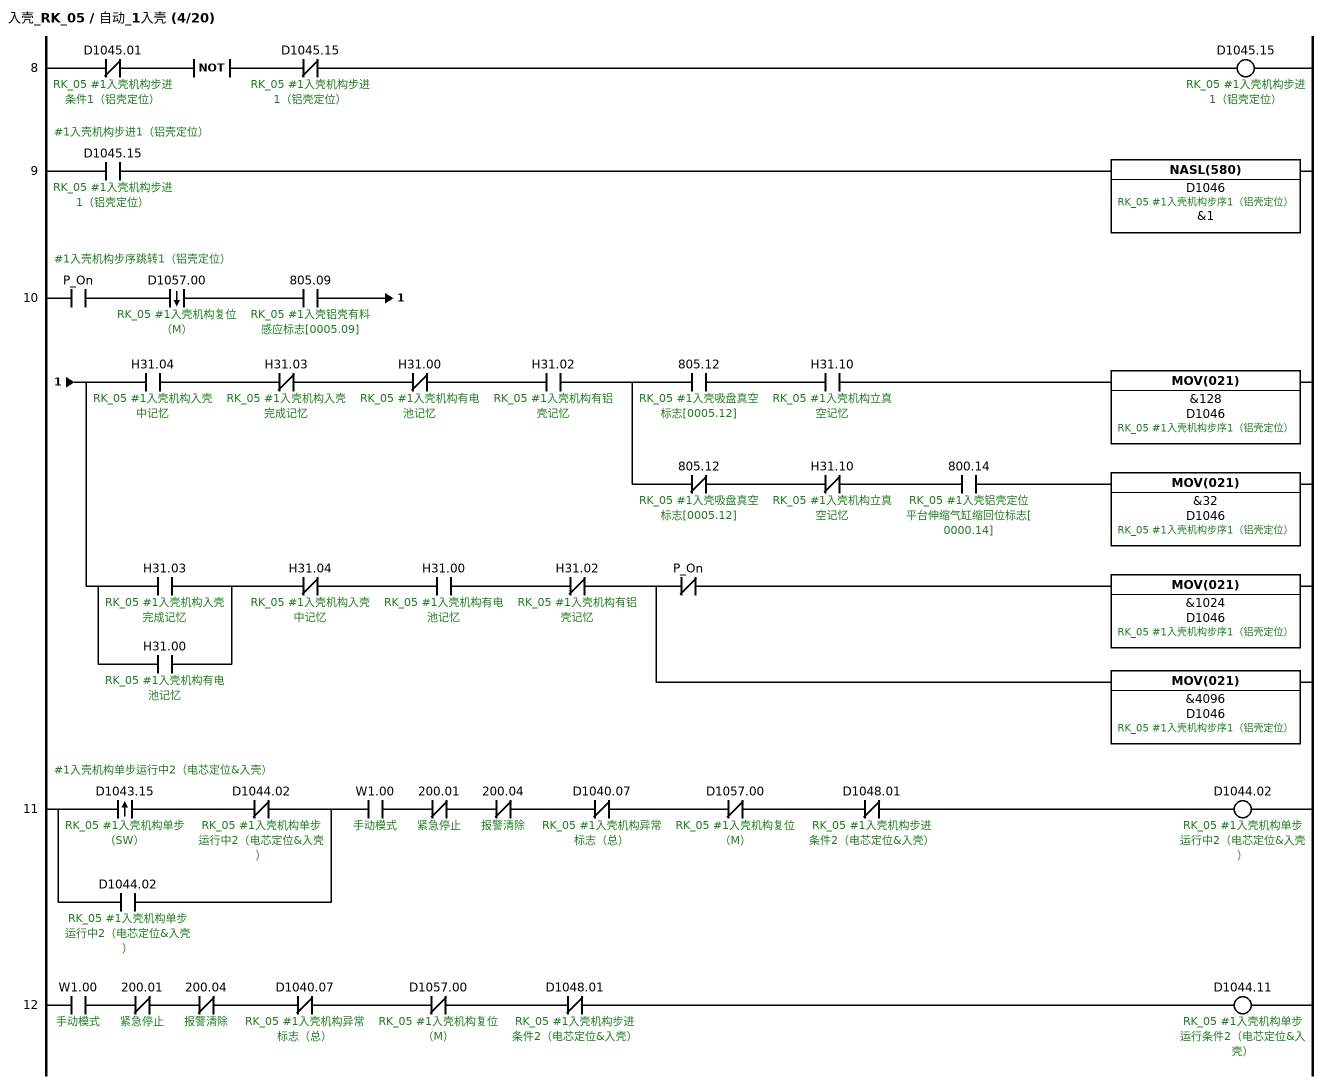
; rung 8
LDNOT D1045.01  ; RK_05 #1入壳机构步进条件1（铝壳定位）
NOT(520)
ANDNOT D1045.15  ; RK_05 #1入壳机构步进1（铝壳定位）
OUT D1045.15  ; RK_05 #1入壳机构步进1（铝壳定位）
; rung 9: #1入壳机构步进1（铝壳定位）
LD D1045.15  ; RK_05 #1入壳机构步进1（铝壳定位）
NASL(580) D1046 &1  ; RK_05 #1入壳机构步序1（铝壳定位）
; rung 10: #1入壳机构步序跳转1（铝壳定位）
LD P_On
%AND D1057.00  ; RK_05 #1入壳机构复位（M）
AND 805.09  ; RK_05 #1入壳铝壳有料感应标志[0005.09]
OUT TR0
AND H31.04  ; RK_05 #1入壳机构入壳中记忆
ANDNOT H31.03  ; RK_05 #1入壳机构入壳完成记忆
ANDNOT H31.00  ; RK_05 #1入壳机构有电池记忆
AND H31.02  ; RK_05 #1入壳机构有铝壳记忆
OUT TR1
AND 805.12  ; RK_05 #1入壳吸盘真空标志[0005.12]
AND H31.10  ; RK_05 #1入壳机构立真空记忆
MOV(021) &128 D1046  ; RK_05 #1入壳机构步序1（铝壳定位）  // RK_05 #1入壳机构吸盘立真空1步（D1046.07）
LD TR1
ANDNOT 805.12  ; RK_05 #1入壳吸盘真空标志[0005.12]
ANDNOT H31.10  ; RK_05 #1入壳机构立真空记忆
AND 800.14  ; RK_05 #1入壳铝壳定位平台伸缩气缸缩回位标志[0000.14]
MOV(021) &32 D1046  ; RK_05 #1入壳机构步序1（铝壳定位）  // RK_05 #1入壳机构铝壳定位平台升降气缸上升1步（D1046.05）
LD TR0
LD H31.03  ; RK_05 #1入壳机构入壳完成记忆
OR H31.00  ; RK_05 #1入壳机构有电池记忆
ANDLD
ANDNOT H31.04  ; RK_05 #1入壳机构入壳中记忆
AND H31.00  ; RK_05 #1入壳机构有电池记忆
ANDNOT H31.02  ; RK_05 #1入壳机构有铝壳记忆
OUT TR0
ANDNOT P_On
MOV(021) &1024 D1046  ; RK_05 #1入壳机构步序1（铝壳定位）  // RK_05 #1入壳机构吸盘破真空&定位陶瓷棒夹紧气缸缩回&铝壳定位平台升降气缸下降1步（D1046.10）
LD TR0
MOV(021) &4096 D1046  ; RK_05 #1入壳机构步序1（铝壳定位）  // RK_05 #1入壳机构铝壳定位平台伸缩气缸伸出1步（D1046.12）
; rung 11: #1入壳机构单步运行中2（电芯定位&入壳）
@LD D1043.15  ; RK_05 #1入壳机构单步（SW）
ANDNOT D1044.02  ; RK_05 #1入壳机构单步运行中2（电芯定位&入壳）
OR D1044.02  ; RK_05 #1入壳机构单步运行中2（电芯定位&入壳）
AND W1.00  ; 手动模式
ANDNOT 200.01  ; 紧急停止
ANDNOT 200.04  ; 报警清除
ANDNOT D1040.07  ; RK_05 #1入壳机构异常标志（总）
ANDNOT D1057.00  ; RK_05 #1入壳机构复位（M）
ANDNOT D1048.01  ; RK_05 #1入壳机构步进条件2（电芯定位&入壳）
OUT D1044.02  ; RK_05 #1入壳机构单步运行中2（电芯定位&入壳）
; rung 12
LD W1.00  ; 手动模式
ANDNOT 200.01  ; 紧急停止
ANDNOT 200.04  ; 报警清除
ANDNOT D1040.07  ; RK_05 #1入壳机构异常标志（总）
ANDNOT D1057.00  ; RK_05 #1入壳机构复位（M）
ANDNOT D1048.01  ; RK_05 #1入壳机构步进条件2（电芯定位&入壳）
OUT D1044.11  ; RK_05 #1入壳机构单步运行条件2（电芯定位&入壳）

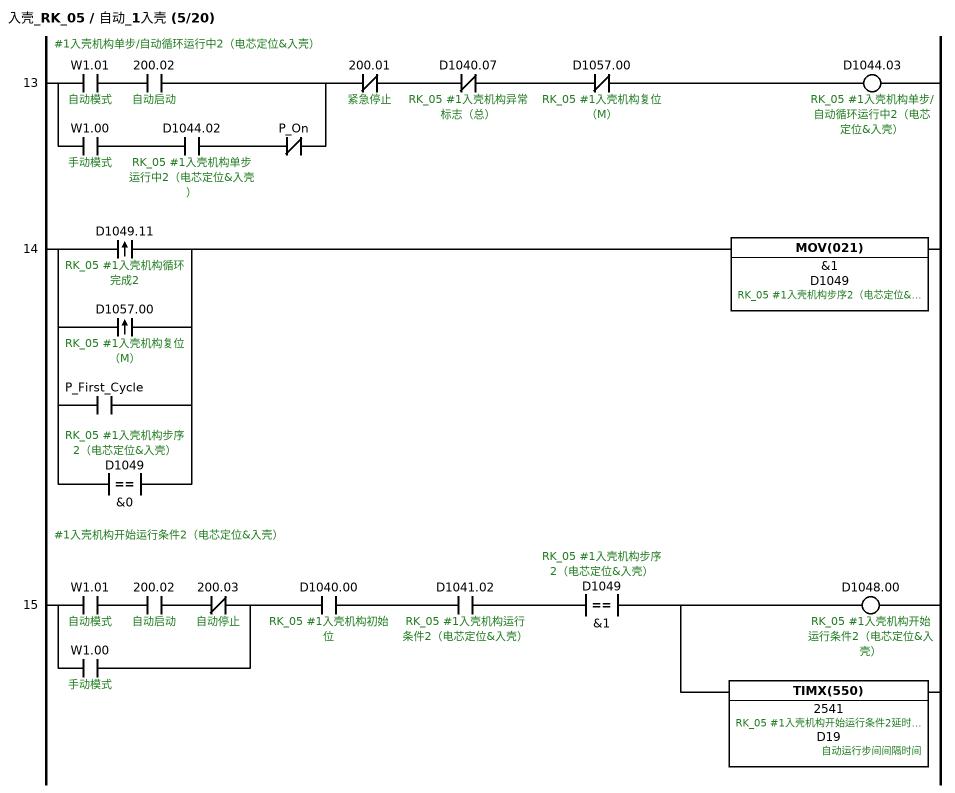
; rung 13: #1入壳机构单步/自动循环运行中2（电芯定位&入壳）
LD W1.01  ; 自动模式
AND 200.02  ; 自动启动
LD W1.00  ; 手动模式
AND D1044.02  ; RK_05 #1入壳机构单步运行中2（电芯定位&入壳）
ANDNOT P_On
ORLD
ANDNOT 200.01  ; 紧急停止
ANDNOT D1040.07  ; RK_05 #1入壳机构异常标志（总）
ANDNOT D1057.00  ; RK_05 #1入壳机构复位（M）
OUT D1044.03  ; RK_05 #1入壳机构单步/自动循环运行中2（电芯定位&入壳）
; rung 14
@LD D1049.11  ; RK_05 #1入壳机构循环完成2
@OR D1057.00  ; RK_05 #1入壳机构复位（M）
OR P_First_Cycle
OR=(300) D1049 &0  ; RK_05 #1入壳机构步序2（电芯定位&入壳）
MOV(021) &1 D1049  ; RK_05 #1入壳机构步序2（电芯定位&入壳）
; rung 15: #1入壳机构开始运行条件2（电芯定位&入壳）
LD W1.01  ; 自动模式
AND 200.02  ; 自动启动
ANDNOT 200.03  ; 自动停止
OR W1.00  ; 手动模式
AND D1040.00  ; RK_05 #1入壳机构初始位
AND D1041.02  ; RK_05 #1入壳机构运行条件2（电芯定位&入壳）
AND=(300) D1049 &1  ; RK_05 #1入壳机构步序2（电芯定位&入壳）
OUT D1048.00  ; RK_05 #1入壳机构开始运行条件2（电芯定位&入壳）
TIMX(550) 2541 D19  ; 自动运行步间间隔时间, RK_05 #1入壳机构开始运行条件2延时（电芯定位&入壳）

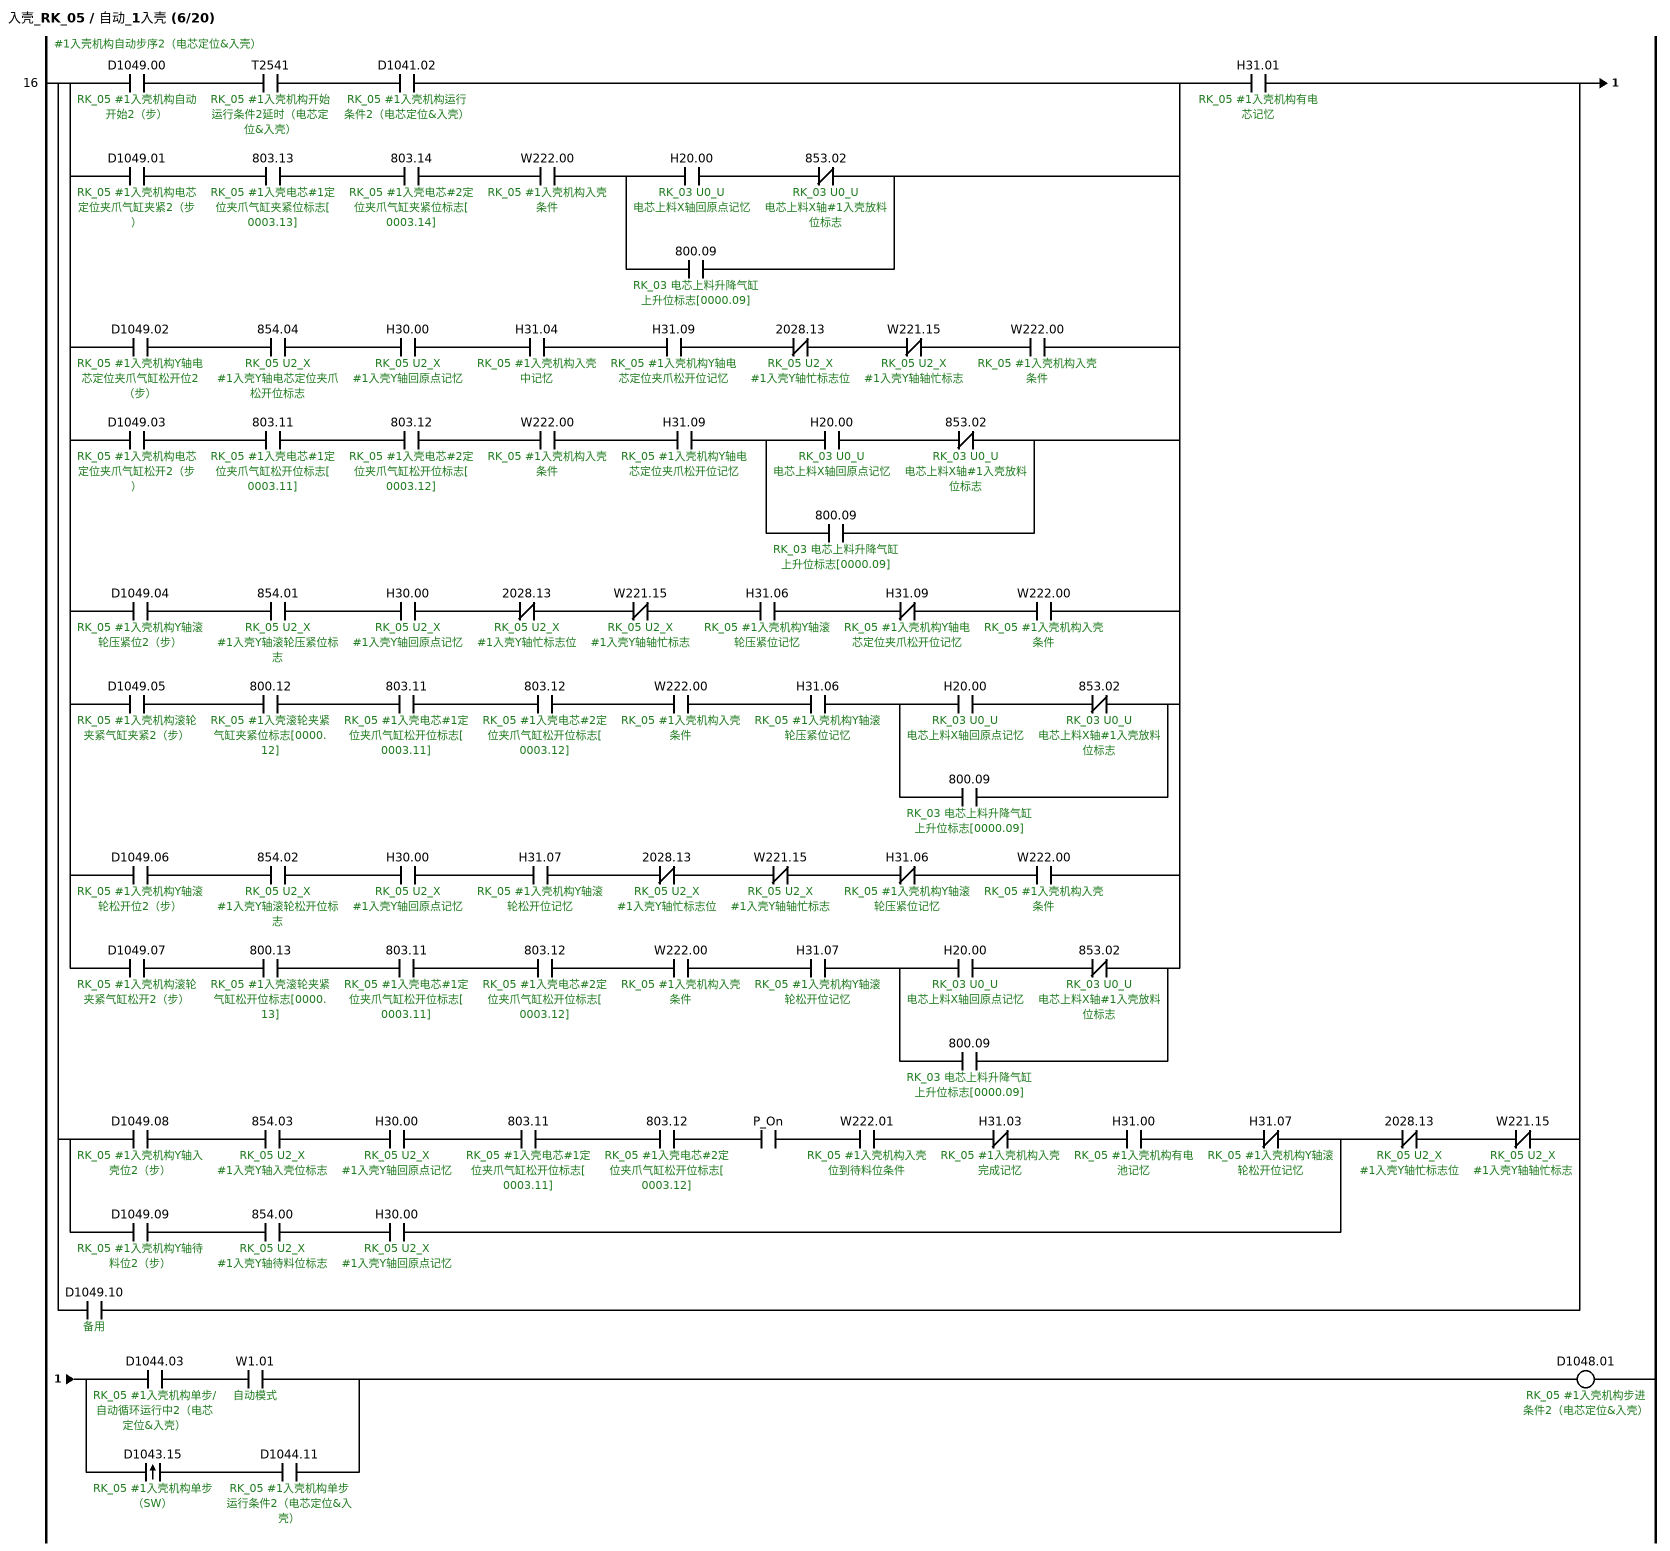
; rung 16: #1入壳机构自动步序2（电芯定位&入壳）
LD D1049.00  ; RK_05 #1入壳机构自动开始2（步）
AND T2541  ; RK_05 #1入壳机构开始运行条件2延时（电芯定位&入壳）
AND D1041.02  ; RK_05 #1入壳机构运行条件2（电芯定位&入壳）
LD D1049.01  ; RK_05 #1入壳机构电芯定位夹爪气缸夹紧2（步）
AND 803.13  ; RK_05 #1入壳电芯#1定位夹爪气缸夹紧位标志[0003.13]
AND 803.14  ; RK_05 #1入壳电芯#2定位夹爪气缸夹紧位标志[0003.14]
AND W222.00  ; RK_05 #1入壳机构入壳条件
LD H20.00  ; RK_03 U0_U 电芯上料X轴回原点记忆
ANDNOT 853.02  ; RK_03 U0_U 电芯上料X轴#1入壳放料位标志
OR 800.09  ; RK_03 电芯上料升降气缸上升位标志[0000.09]
ANDLD
ORLD
LD D1049.02  ; RK_05 #1入壳机构Y轴电芯定位夹爪气缸松开位2（步）
AND 854.04  ; RK_05 U2_X #1入壳Y轴电芯定位夹爪松开位标志
AND H30.00  ; RK_05 U2_X #1入壳Y轴回原点记忆
AND H31.04  ; RK_05 #1入壳机构入壳中记忆
AND H31.09  ; RK_05 #1入壳机构Y轴电芯定位夹爪松开位记忆
ANDNOT 2028.13  ; RK_05 U2_X #1入壳Y轴忙标志位
ANDNOT W221.15  ; RK_05 U2_X #1入壳Y轴轴忙标志
AND W222.00  ; RK_05 #1入壳机构入壳条件
ORLD
LD D1049.03  ; RK_05 #1入壳机构电芯定位夹爪气缸松开2（步）
AND 803.11  ; RK_05 #1入壳电芯#1定位夹爪气缸松开位标志[0003.11]
AND 803.12  ; RK_05 #1入壳电芯#2定位夹爪气缸松开位标志[0003.12]
AND W222.00  ; RK_05 #1入壳机构入壳条件
AND H31.09  ; RK_05 #1入壳机构Y轴电芯定位夹爪松开位记忆
LD H20.00  ; RK_03 U0_U 电芯上料X轴回原点记忆
ANDNOT 853.02  ; RK_03 U0_U 电芯上料X轴#1入壳放料位标志
OR 800.09  ; RK_03 电芯上料升降气缸上升位标志[0000.09]
ANDLD
ORLD
LD D1049.04  ; RK_05 #1入壳机构Y轴滚轮压紧位2（步）
AND 854.01  ; RK_05 U2_X #1入壳Y轴滚轮压紧位标志
AND H30.00  ; RK_05 U2_X #1入壳Y轴回原点记忆
ANDNOT 2028.13  ; RK_05 U2_X #1入壳Y轴忙标志位
ANDNOT W221.15  ; RK_05 U2_X #1入壳Y轴轴忙标志
AND H31.06  ; RK_05 #1入壳机构Y轴滚轮压紧位记忆
ANDNOT H31.09  ; RK_05 #1入壳机构Y轴电芯定位夹爪松开位记忆
AND W222.00  ; RK_05 #1入壳机构入壳条件
ORLD
LD D1049.05  ; RK_05 #1入壳机构滚轮夹紧气缸夹紧2（步）
AND 800.12  ; RK_05 #1入壳滚轮夹紧气缸夹紧位标志[0000.12]
AND 803.11  ; RK_05 #1入壳电芯#1定位夹爪气缸松开位标志[0003.11]
AND 803.12  ; RK_05 #1入壳电芯#2定位夹爪气缸松开位标志[0003.12]
AND W222.00  ; RK_05 #1入壳机构入壳条件
AND H31.06  ; RK_05 #1入壳机构Y轴滚轮压紧位记忆
LD H20.00  ; RK_03 U0_U 电芯上料X轴回原点记忆
ANDNOT 853.02  ; RK_03 U0_U 电芯上料X轴#1入壳放料位标志
OR 800.09  ; RK_03 电芯上料升降气缸上升位标志[0000.09]
ANDLD
ORLD
LD D1049.06  ; RK_05 #1入壳机构Y轴滚轮松开位2（步）
AND 854.02  ; RK_05 U2_X #1入壳Y轴滚轮松开位标志
AND H30.00  ; RK_05 U2_X #1入壳Y轴回原点记忆
AND H31.07  ; RK_05 #1入壳机构Y轴滚轮松开位记忆
ANDNOT 2028.13  ; RK_05 U2_X #1入壳Y轴忙标志位
ANDNOT W221.15  ; RK_05 U2_X #1入壳Y轴轴忙标志
ANDNOT H31.06  ; RK_05 #1入壳机构Y轴滚轮压紧位记忆
AND W222.00  ; RK_05 #1入壳机构入壳条件
ORLD
LD D1049.07  ; RK_05 #1入壳机构滚轮夹紧气缸松开2（步）
AND 800.13  ; RK_05 #1入壳滚轮夹紧气缸松开位标志[0000.13]
AND 803.11  ; RK_05 #1入壳电芯#1定位夹爪气缸松开位标志[0003.11]
AND 803.12  ; RK_05 #1入壳电芯#2定位夹爪气缸松开位标志[0003.12]
AND W222.00  ; RK_05 #1入壳机构入壳条件
AND H31.07  ; RK_05 #1入壳机构Y轴滚轮松开位记忆
LD H20.00  ; RK_03 U0_U 电芯上料X轴回原点记忆
ANDNOT 853.02  ; RK_03 U0_U 电芯上料X轴#1入壳放料位标志
OR 800.09  ; RK_03 电芯上料升降气缸上升位标志[0000.09]
ANDLD
ORLD
AND H31.01  ; RK_05 #1入壳机构有电芯记忆
LD D1049.08  ; RK_05 #1入壳机构Y轴入壳位2（步）
AND 854.03  ; RK_05 U2_X #1入壳Y轴入壳位标志
AND H30.00  ; RK_05 U2_X #1入壳Y轴回原点记忆
AND 803.11  ; RK_05 #1入壳电芯#1定位夹爪气缸松开位标志[0003.11]
AND 803.12  ; RK_05 #1入壳电芯#2定位夹爪气缸松开位标志[0003.12]
AND P_On  // 是否增加到入壳位后稳定延时？
AND W222.01  ; RK_05 #1入壳机构入壳位到待料位条件
ANDNOT H31.03  ; RK_05 #1入壳机构入壳完成记忆
AND H31.00  ; RK_05 #1入壳机构有电池记忆
ANDNOT H31.07  ; RK_05 #1入壳机构Y轴滚轮松开位记忆
LD D1049.09  ; RK_05 #1入壳机构Y轴待料位2（步）
AND 854.00  ; RK_05 U2_X #1入壳Y轴待料位标志
AND H30.00  ; RK_05 U2_X #1入壳Y轴回原点记忆
ORLD
ANDNOT 2028.13  ; RK_05 U2_X #1入壳Y轴忙标志位
ANDNOT W221.15  ; RK_05 U2_X #1入壳Y轴轴忙标志
ORLD
OR D1049.10  ; 备用
LD D1044.03  ; RK_05 #1入壳机构单步/自动循环运行中2（电芯定位&入壳）
AND W1.01  ; 自动模式
@LD D1043.15  ; RK_05 #1入壳机构单步（SW）
AND D1044.11  ; RK_05 #1入壳机构单步运行条件2（电芯定位&入壳）
ORLD
ANDLD
OUT D1048.01  ; RK_05 #1入壳机构步进条件2（电芯定位&入壳）

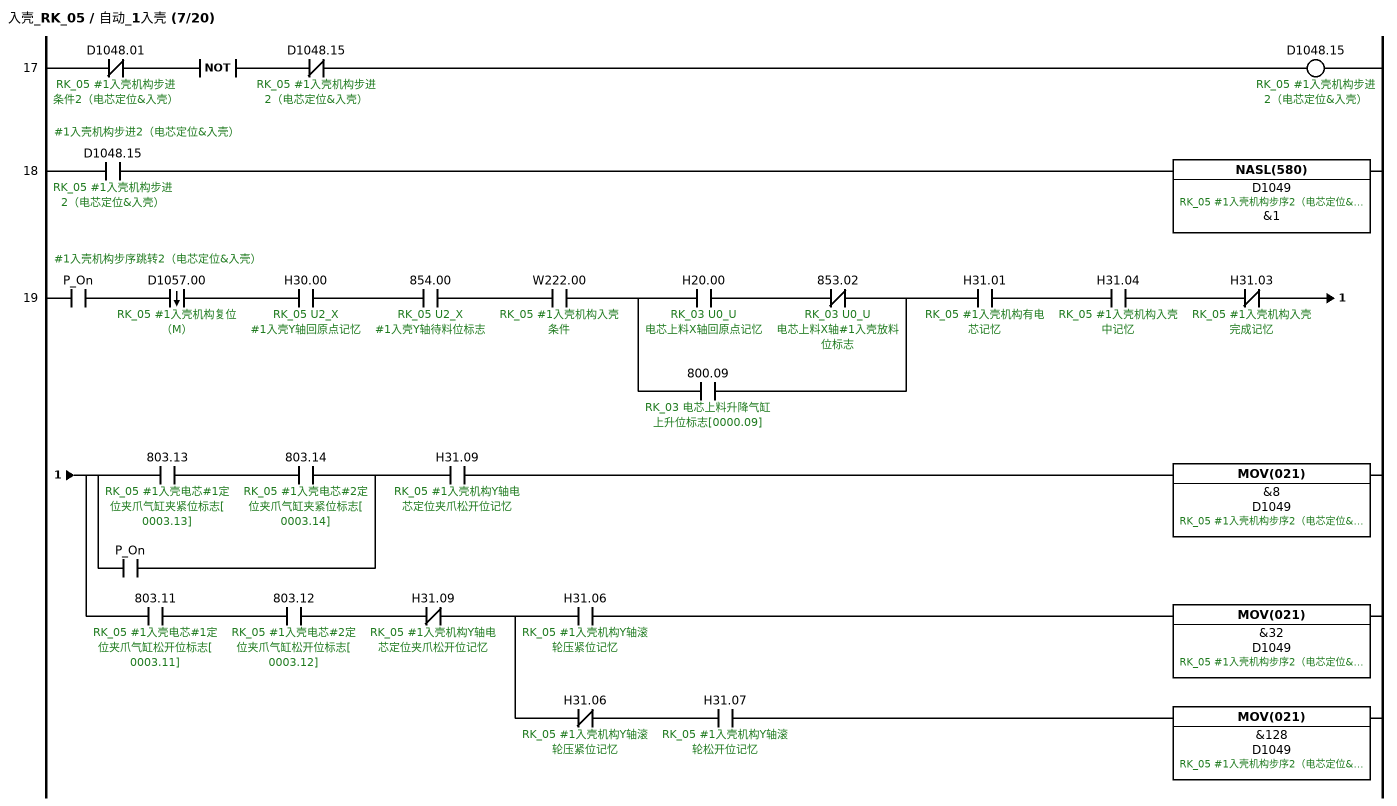
; rung 17
LDNOT D1048.01  ; RK_05 #1入壳机构步进条件2（电芯定位&入壳）
NOT(520)
ANDNOT D1048.15  ; RK_05 #1入壳机构步进2（电芯定位&入壳）
OUT D1048.15  ; RK_05 #1入壳机构步进2（电芯定位&入壳）
; rung 18: #1入壳机构步进2（电芯定位&入壳）
LD D1048.15  ; RK_05 #1入壳机构步进2（电芯定位&入壳）
NASL(580) D1049 &1  ; RK_05 #1入壳机构步序2（电芯定位&入壳）
; rung 19: #1入壳机构步序跳转2（电芯定位&入壳）
LD P_On
%AND D1057.00  ; RK_05 #1入壳机构复位（M）
AND H30.00  ; RK_05 U2_X #1入壳Y轴回原点记忆
AND 854.00  ; RK_05 U2_X #1入壳Y轴待料位标志
AND W222.00  ; RK_05 #1入壳机构入壳条件
LD H20.00  ; RK_03 U0_U 电芯上料X轴回原点记忆
ANDNOT 853.02  ; RK_03 U0_U 电芯上料X轴#1入壳放料位标志
OR 800.09  ; RK_03 电芯上料升降气缸上升位标志[0000.09]
ANDLD
AND H31.01  ; RK_05 #1入壳机构有电芯记忆
AND H31.04  ; RK_05 #1入壳机构入壳中记忆
ANDNOT H31.03  ; RK_05 #1入壳机构入壳完成记忆
OUT TR0
LD 803.13  ; RK_05 #1入壳电芯#1定位夹爪气缸夹紧位标志[0003.13]
AND 803.14  ; RK_05 #1入壳电芯#2定位夹爪气缸夹紧位标志[0003.14]
OR P_On
ANDLD
AND H31.09  ; RK_05 #1入壳机构Y轴电芯定位夹爪松开位记忆
MOV(021) &8 D1049  ; RK_05 #1入壳机构步序2（电芯定位&入壳）  // RK_05 #1入壳机构电芯定位夹爪气缸松开2步（D1049.03）
LD TR0
AND 803.11  ; RK_05 #1入壳电芯#1定位夹爪气缸松开位标志[0003.11]
AND 803.12  ; RK_05 #1入壳电芯#2定位夹爪气缸松开位标志[0003.12]
ANDNOT H31.09  ; RK_05 #1入壳机构Y轴电芯定位夹爪松开位记忆
OUT TR0
AND H31.06  ; RK_05 #1入壳机构Y轴滚轮压紧位记忆
MOV(021) &32 D1049  ; RK_05 #1入壳机构步序2（电芯定位&入壳）  // RK_05 #1入壳机构滚轮夹紧气缸夹紧2步（D1049.05）
LD TR0
ANDNOT H31.06  ; RK_05 #1入壳机构Y轴滚轮压紧位记忆
AND H31.07  ; RK_05 #1入壳机构Y轴滚轮松开位记忆
MOV(021) &128 D1049  ; RK_05 #1入壳机构步序2（电芯定位&入壳）  // RK_05 #1入壳机构滚轮夹紧气缸松开2步（D1049.07）

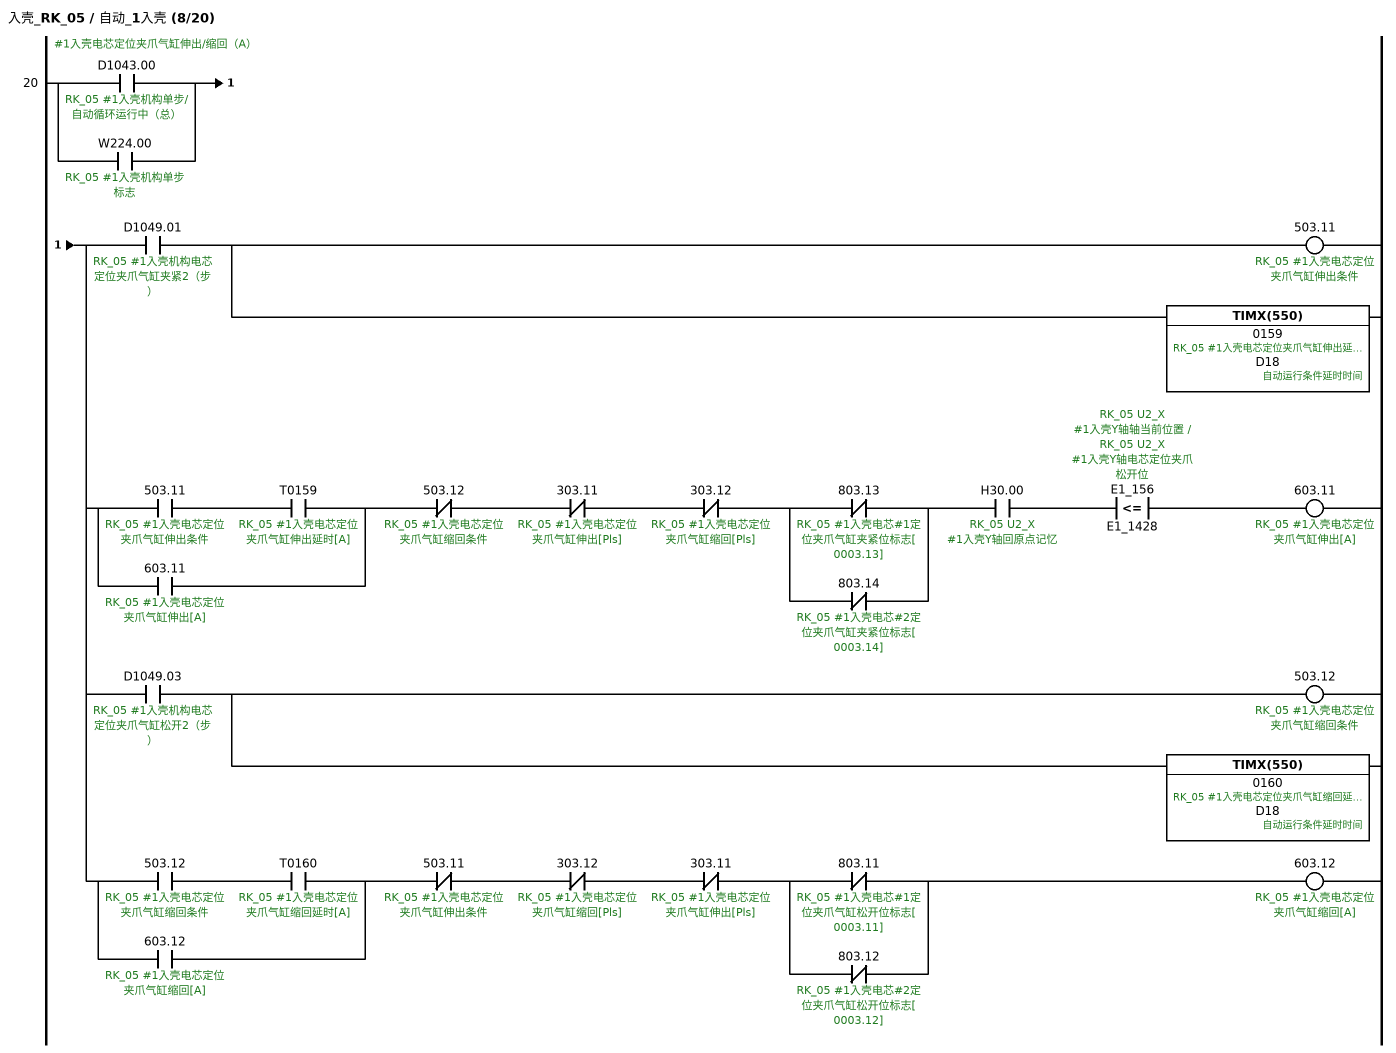
; rung 20: #1入壳电芯定位夹爪气缸伸出/缩回（A）
LD D1043.00  ; RK_05 #1入壳机构单步/自动循环运行中（总）
OR W224.00  ; RK_05 #1入壳机构单步标志
OUT TR0
AND D1049.01  ; RK_05 #1入壳机构电芯定位夹爪气缸夹紧2（步）
OUT 503.11  ; RK_05 #1入壳电芯定位夹爪气缸伸出条件
TIMX(550) 0159 D18  ; 自动运行条件延时时间, RK_05 #1入壳电芯定位夹爪气缸伸出延时[A]
LD TR0
LD 503.11  ; RK_05 #1入壳电芯定位夹爪气缸伸出条件
AND T0159  ; RK_05 #1入壳电芯定位夹爪气缸伸出延时[A]
OR 603.11  ; RK_05 #1入壳电芯定位夹爪气缸伸出[A]
ANDLD
ANDNOT 503.12  ; RK_05 #1入壳电芯定位夹爪气缸缩回条件
ANDNOT 303.11  ; RK_05 #1入壳电芯定位夹爪气缸伸出[Pls]
ANDNOT 303.12  ; RK_05 #1入壳电芯定位夹爪气缸缩回[Pls]
LDNOT 803.13  ; RK_05 #1入壳电芯#1定位夹爪气缸夹紧位标志[0003.13]
ORNOT 803.14  ; RK_05 #1入壳电芯#2定位夹爪气缸夹紧位标志[0003.14]
ANDLD
AND H30.00  ; RK_05 U2_X #1入壳Y轴回原点记忆
AND<=SL(318) E1_156 E1_1428  ; RK_05 U2_X #1入壳Y轴轴当前位置, RK_05 U2_X #1入壳Y轴电芯定位夹爪松开位
OUT 603.11  ; RK_05 #1入壳电芯定位夹爪气缸伸出[A]
LD TR0
AND D1049.03  ; RK_05 #1入壳机构电芯定位夹爪气缸松开2（步）
OUT 503.12  ; RK_05 #1入壳电芯定位夹爪气缸缩回条件
TIMX(550) 0160 D18  ; 自动运行条件延时时间, RK_05 #1入壳电芯定位夹爪气缸缩回延时[A]
LD TR0
LD 503.12  ; RK_05 #1入壳电芯定位夹爪气缸缩回条件
AND T0160  ; RK_05 #1入壳电芯定位夹爪气缸缩回延时[A]
OR 603.12  ; RK_05 #1入壳电芯定位夹爪气缸缩回[A]
ANDLD
ANDNOT 503.11  ; RK_05 #1入壳电芯定位夹爪气缸伸出条件
ANDNOT 303.12  ; RK_05 #1入壳电芯定位夹爪气缸缩回[Pls]
ANDNOT 303.11  ; RK_05 #1入壳电芯定位夹爪气缸伸出[Pls]
LDNOT 803.11  ; RK_05 #1入壳电芯#1定位夹爪气缸松开位标志[0003.11]
ORNOT 803.12  ; RK_05 #1入壳电芯#2定位夹爪气缸松开位标志[0003.12]
ANDLD
OUT 603.12  ; RK_05 #1入壳电芯定位夹爪气缸缩回[A]

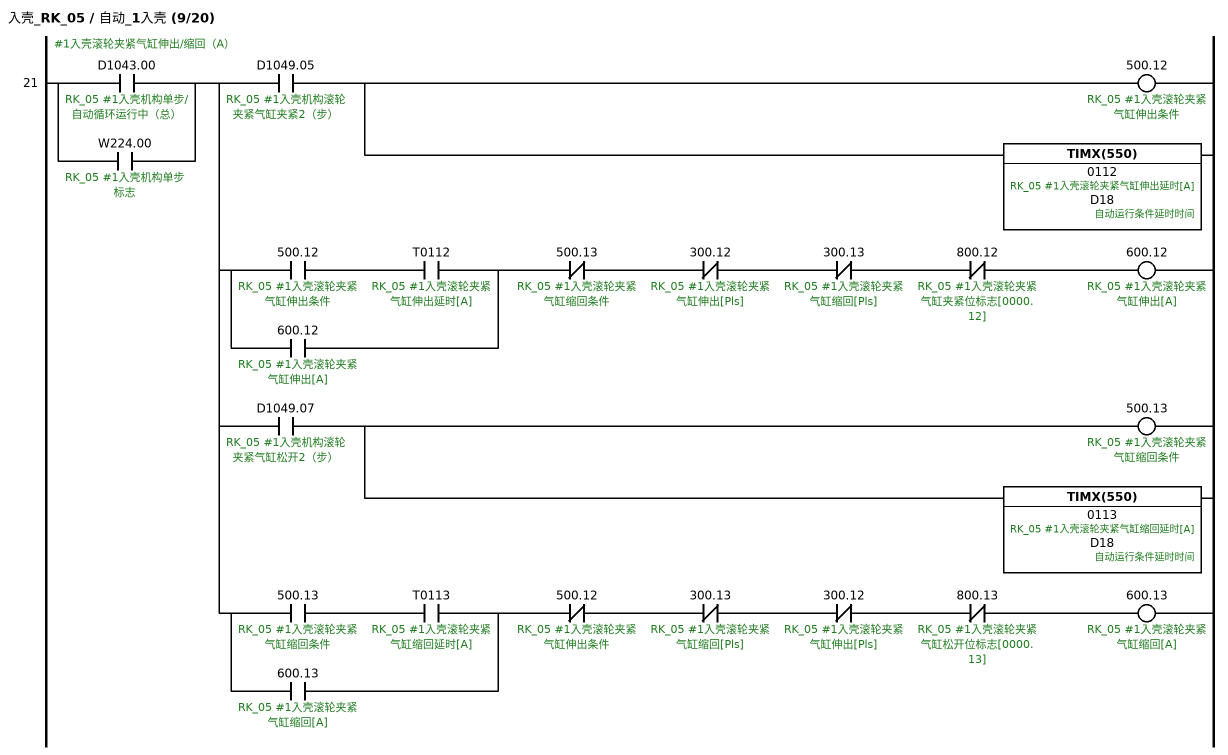
; rung 21: #1入壳滚轮夹紧气缸伸出/缩回（A）
LD D1043.00  ; RK_05 #1入壳机构单步/自动循环运行中（总）
OR W224.00  ; RK_05 #1入壳机构单步标志
OUT TR0
AND D1049.05  ; RK_05 #1入壳机构滚轮夹紧气缸夹紧2（步）
OUT 500.12  ; RK_05 #1入壳滚轮夹紧气缸伸出条件
TIMX(550) 0112 D18  ; 自动运行条件延时时间, RK_05 #1入壳滚轮夹紧气缸伸出延时[A]
LD TR0
LD 500.12  ; RK_05 #1入壳滚轮夹紧气缸伸出条件
AND T0112  ; RK_05 #1入壳滚轮夹紧气缸伸出延时[A]
OR 600.12  ; RK_05 #1入壳滚轮夹紧气缸伸出[A]
ANDLD
ANDNOT 500.13  ; RK_05 #1入壳滚轮夹紧气缸缩回条件
ANDNOT 300.12  ; RK_05 #1入壳滚轮夹紧气缸伸出[Pls]
ANDNOT 300.13  ; RK_05 #1入壳滚轮夹紧气缸缩回[Pls]
ANDNOT 800.12  ; RK_05 #1入壳滚轮夹紧气缸夹紧位标志[0000.12]
OUT 600.12  ; RK_05 #1入壳滚轮夹紧气缸伸出[A]
LD TR0
AND D1049.07  ; RK_05 #1入壳机构滚轮夹紧气缸松开2（步）
OUT 500.13  ; RK_05 #1入壳滚轮夹紧气缸缩回条件
TIMX(550) 0113 D18  ; 自动运行条件延时时间, RK_05 #1入壳滚轮夹紧气缸缩回延时[A]
LD TR0
LD 500.13  ; RK_05 #1入壳滚轮夹紧气缸缩回条件
AND T0113  ; RK_05 #1入壳滚轮夹紧气缸缩回延时[A]
OR 600.13  ; RK_05 #1入壳滚轮夹紧气缸缩回[A]
ANDLD
ANDNOT 500.12  ; RK_05 #1入壳滚轮夹紧气缸伸出条件
ANDNOT 300.13  ; RK_05 #1入壳滚轮夹紧气缸缩回[Pls]
ANDNOT 300.12  ; RK_05 #1入壳滚轮夹紧气缸伸出[Pls]
ANDNOT 800.13  ; RK_05 #1入壳滚轮夹紧气缸松开位标志[0000.13]
OUT 600.13  ; RK_05 #1入壳滚轮夹紧气缸缩回[A]

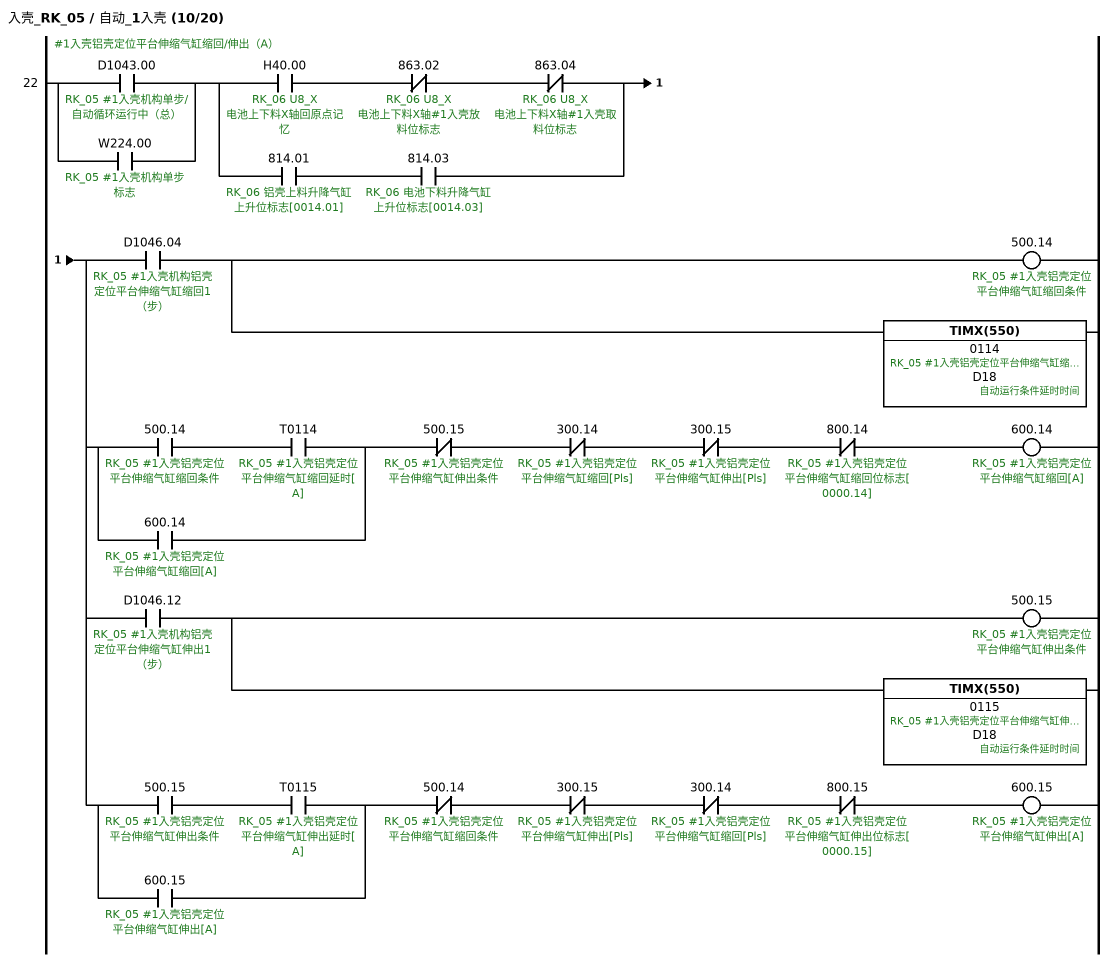
; rung 22: #1入壳铝壳定位平台伸缩气缸缩回/伸出（A）
LD D1043.00  ; RK_05 #1入壳机构单步/自动循环运行中（总）
OR W224.00  ; RK_05 #1入壳机构单步标志
LD H40.00  ; RK_06 U8_X 电池上下料X轴回原点记忆
ANDNOT 863.02  ; RK_06 U8_X 电池上下料X轴#1入壳放料位标志
ANDNOT 863.04  ; RK_06 U8_X 电池上下料X轴#1入壳取料位标志
LD 814.01  ; RK_06 铝壳上料升降气缸上升位标志[0014.01]
AND 814.03  ; RK_06 电池下料升降气缸上升位标志[0014.03]
ORLD
ANDLD
OUT TR0
AND D1046.04  ; RK_05 #1入壳机构铝壳定位平台伸缩气缸缩回1（步）
OUT 500.14  ; RK_05 #1入壳铝壳定位平台伸缩气缸缩回条件
TIMX(550) 0114 D18  ; 自动运行条件延时时间, RK_05 #1入壳铝壳定位平台伸缩气缸缩回延时[A]
LD TR0
LD 500.14  ; RK_05 #1入壳铝壳定位平台伸缩气缸缩回条件
AND T0114  ; RK_05 #1入壳铝壳定位平台伸缩气缸缩回延时[A]
OR 600.14  ; RK_05 #1入壳铝壳定位平台伸缩气缸缩回[A]
ANDLD
ANDNOT 500.15  ; RK_05 #1入壳铝壳定位平台伸缩气缸伸出条件
ANDNOT 300.14  ; RK_05 #1入壳铝壳定位平台伸缩气缸缩回[Pls]
ANDNOT 300.15  ; RK_05 #1入壳铝壳定位平台伸缩气缸伸出[Pls]
ANDNOT 800.14  ; RK_05 #1入壳铝壳定位平台伸缩气缸缩回位标志[0000.14]
OUT 600.14  ; RK_05 #1入壳铝壳定位平台伸缩气缸缩回[A]
LD TR0
AND D1046.12  ; RK_05 #1入壳机构铝壳定位平台伸缩气缸伸出1（步）
OUT 500.15  ; RK_05 #1入壳铝壳定位平台伸缩气缸伸出条件
TIMX(550) 0115 D18  ; 自动运行条件延时时间, RK_05 #1入壳铝壳定位平台伸缩气缸伸出延时[A]
LD TR0
LD 500.15  ; RK_05 #1入壳铝壳定位平台伸缩气缸伸出条件
AND T0115  ; RK_05 #1入壳铝壳定位平台伸缩气缸伸出延时[A]
OR 600.15  ; RK_05 #1入壳铝壳定位平台伸缩气缸伸出[A]
ANDLD
ANDNOT 500.14  ; RK_05 #1入壳铝壳定位平台伸缩气缸缩回条件
ANDNOT 300.15  ; RK_05 #1入壳铝壳定位平台伸缩气缸伸出[Pls]
ANDNOT 300.14  ; RK_05 #1入壳铝壳定位平台伸缩气缸缩回[Pls]
ANDNOT 800.15  ; RK_05 #1入壳铝壳定位平台伸缩气缸伸出位标志[0000.15]
OUT 600.15  ; RK_05 #1入壳铝壳定位平台伸缩气缸伸出[A]

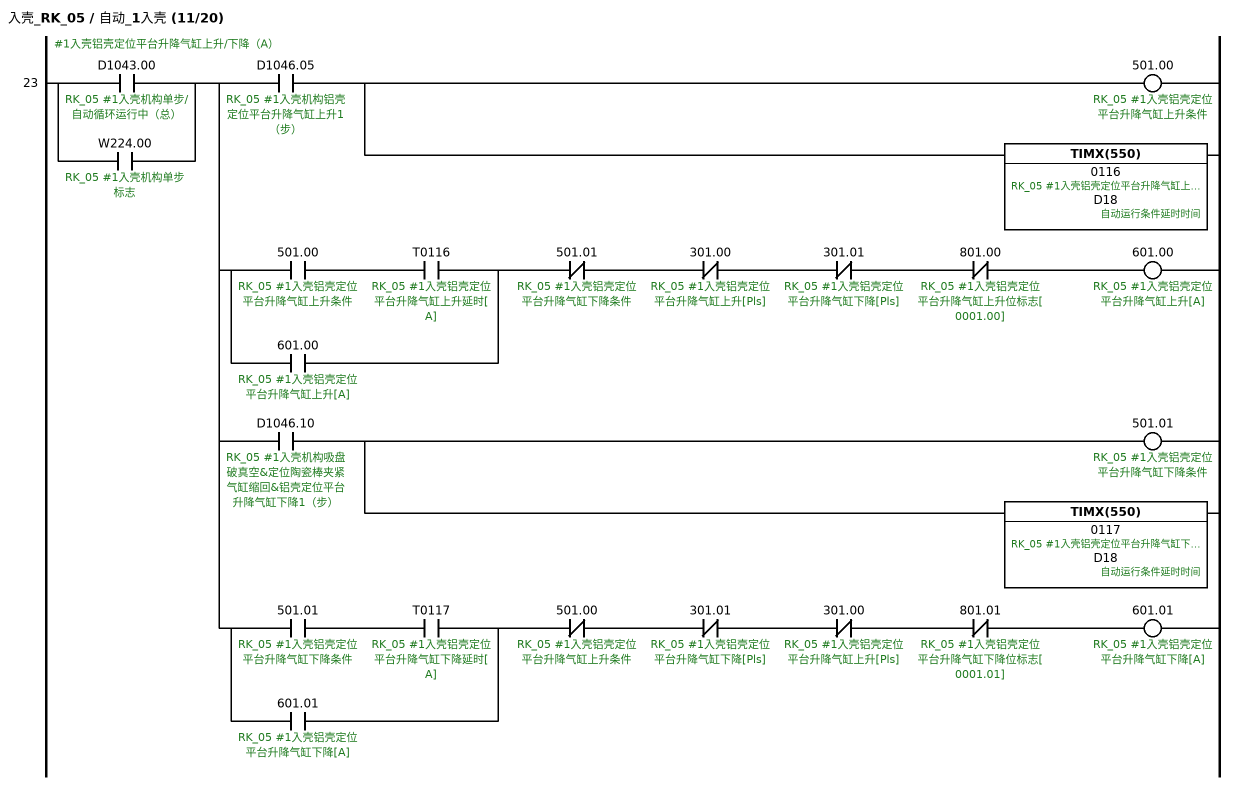
; rung 23: #1入壳铝壳定位平台升降气缸上升/下降（A）
LD D1043.00  ; RK_05 #1入壳机构单步/自动循环运行中（总）
OR W224.00  ; RK_05 #1入壳机构单步标志
OUT TR0
AND D1046.05  ; RK_05 #1入壳机构铝壳定位平台升降气缸上升1（步）
OUT 501.00  ; RK_05 #1入壳铝壳定位平台升降气缸上升条件
TIMX(550) 0116 D18  ; 自动运行条件延时时间, RK_05 #1入壳铝壳定位平台升降气缸上升延时[A]
LD TR0
LD 501.00  ; RK_05 #1入壳铝壳定位平台升降气缸上升条件
AND T0116  ; RK_05 #1入壳铝壳定位平台升降气缸上升延时[A]
OR 601.00  ; RK_05 #1入壳铝壳定位平台升降气缸上升[A]
ANDLD
ANDNOT 501.01  ; RK_05 #1入壳铝壳定位平台升降气缸下降条件
ANDNOT 301.00  ; RK_05 #1入壳铝壳定位平台升降气缸上升[Pls]
ANDNOT 301.01  ; RK_05 #1入壳铝壳定位平台升降气缸下降[Pls]
ANDNOT 801.00  ; RK_05 #1入壳铝壳定位平台升降气缸上升位标志[0001.00]
OUT 601.00  ; RK_05 #1入壳铝壳定位平台升降气缸上升[A]
LD TR0
AND D1046.10  ; RK_05 #1入壳机构吸盘破真空&定位陶瓷棒夹紧气缸缩回&铝壳定位平台升降气缸下降1（步）
OUT 501.01  ; RK_05 #1入壳铝壳定位平台升降气缸下降条件
TIMX(550) 0117 D18  ; 自动运行条件延时时间, RK_05 #1入壳铝壳定位平台升降气缸下降延时[A]
LD TR0
LD 501.01  ; RK_05 #1入壳铝壳定位平台升降气缸下降条件
AND T0117  ; RK_05 #1入壳铝壳定位平台升降气缸下降延时[A]
OR 601.01  ; RK_05 #1入壳铝壳定位平台升降气缸下降[A]
ANDLD
ANDNOT 501.00  ; RK_05 #1入壳铝壳定位平台升降气缸上升条件
ANDNOT 301.01  ; RK_05 #1入壳铝壳定位平台升降气缸下降[Pls]
ANDNOT 301.00  ; RK_05 #1入壳铝壳定位平台升降气缸上升[Pls]
ANDNOT 801.01  ; RK_05 #1入壳铝壳定位平台升降气缸下降位标志[0001.01]
OUT 601.01  ; RK_05 #1入壳铝壳定位平台升降气缸下降[A]

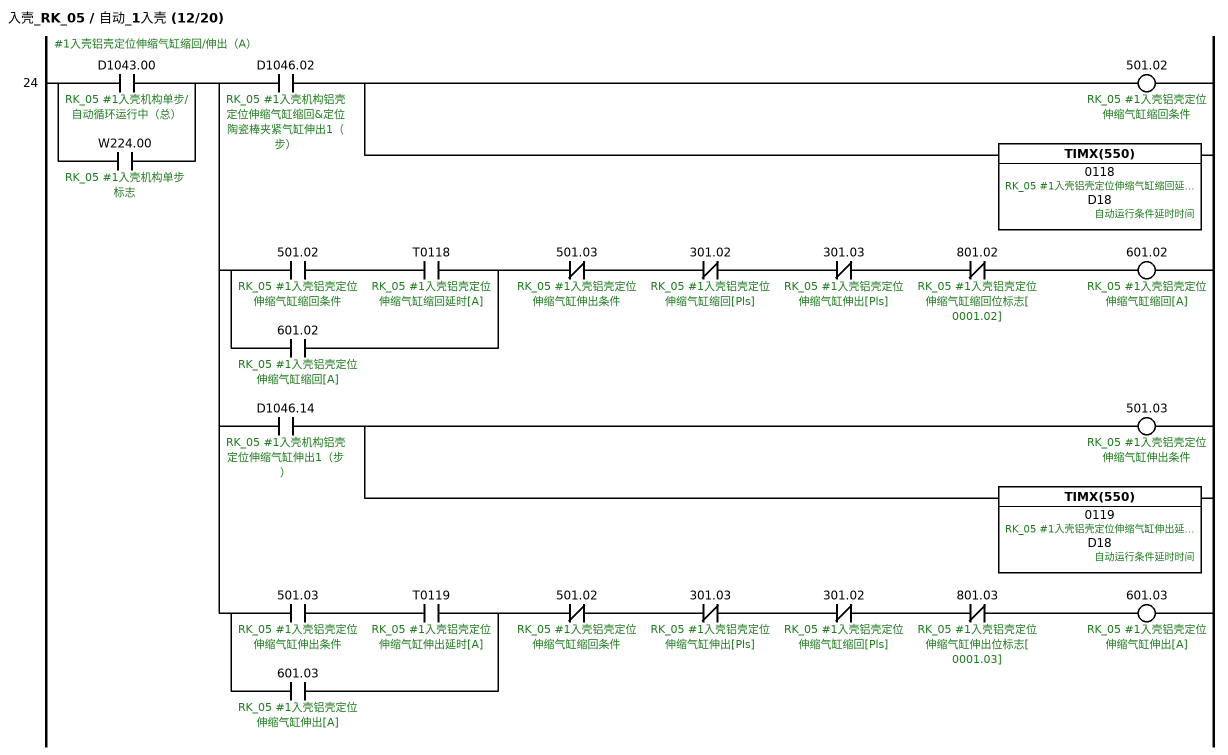
; rung 24: #1入壳铝壳定位伸缩气缸缩回/伸出（A）
LD D1043.00  ; RK_05 #1入壳机构单步/自动循环运行中（总）
OR W224.00  ; RK_05 #1入壳机构单步标志
OUT TR0
AND D1046.02  ; RK_05 #1入壳机构铝壳定位伸缩气缸缩回&定位陶瓷棒夹紧气缸伸出1（步）
OUT 501.02  ; RK_05 #1入壳铝壳定位伸缩气缸缩回条件
TIMX(550) 0118 D18  ; 自动运行条件延时时间, RK_05 #1入壳铝壳定位伸缩气缸缩回延时[A]
LD TR0
LD 501.02  ; RK_05 #1入壳铝壳定位伸缩气缸缩回条件
AND T0118  ; RK_05 #1入壳铝壳定位伸缩气缸缩回延时[A]
OR 601.02  ; RK_05 #1入壳铝壳定位伸缩气缸缩回[A]
ANDLD
ANDNOT 501.03  ; RK_05 #1入壳铝壳定位伸缩气缸伸出条件
ANDNOT 301.02  ; RK_05 #1入壳铝壳定位伸缩气缸缩回[Pls]
ANDNOT 301.03  ; RK_05 #1入壳铝壳定位伸缩气缸伸出[Pls]
ANDNOT 801.02  ; RK_05 #1入壳铝壳定位伸缩气缸缩回位标志[0001.02]
OUT 601.02  ; RK_05 #1入壳铝壳定位伸缩气缸缩回[A]
LD TR0
AND D1046.14  ; RK_05 #1入壳机构铝壳定位伸缩气缸伸出1（步）
OUT 501.03  ; RK_05 #1入壳铝壳定位伸缩气缸伸出条件
TIMX(550) 0119 D18  ; 自动运行条件延时时间, RK_05 #1入壳铝壳定位伸缩气缸伸出延时[A]
LD TR0
LD 501.03  ; RK_05 #1入壳铝壳定位伸缩气缸伸出条件
AND T0119  ; RK_05 #1入壳铝壳定位伸缩气缸伸出延时[A]
OR 601.03  ; RK_05 #1入壳铝壳定位伸缩气缸伸出[A]
ANDLD
ANDNOT 501.02  ; RK_05 #1入壳铝壳定位伸缩气缸缩回条件
ANDNOT 301.03  ; RK_05 #1入壳铝壳定位伸缩气缸伸出[Pls]
ANDNOT 301.02  ; RK_05 #1入壳铝壳定位伸缩气缸缩回[Pls]
ANDNOT 801.03  ; RK_05 #1入壳铝壳定位伸缩气缸伸出位标志[0001.03]
OUT 601.03  ; RK_05 #1入壳铝壳定位伸缩气缸伸出[A]

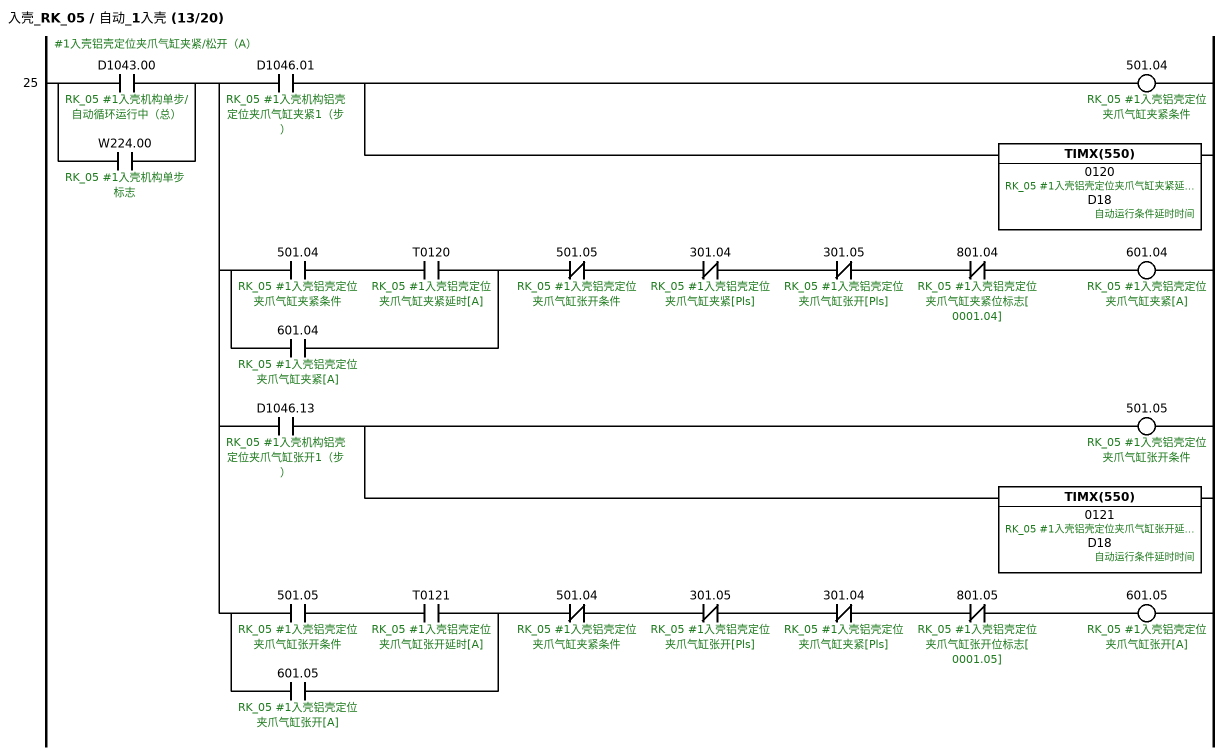
; rung 25: #1入壳铝壳定位夹爪气缸夹紧/松开（A）
LD D1043.00  ; RK_05 #1入壳机构单步/自动循环运行中（总）
OR W224.00  ; RK_05 #1入壳机构单步标志
OUT TR0
AND D1046.01  ; RK_05 #1入壳机构铝壳定位夹爪气缸夹紧1（步）
OUT 501.04  ; RK_05 #1入壳铝壳定位夹爪气缸夹紧条件
TIMX(550) 0120 D18  ; 自动运行条件延时时间, RK_05 #1入壳铝壳定位夹爪气缸夹紧延时[A]
LD TR0
LD 501.04  ; RK_05 #1入壳铝壳定位夹爪气缸夹紧条件
AND T0120  ; RK_05 #1入壳铝壳定位夹爪气缸夹紧延时[A]
OR 601.04  ; RK_05 #1入壳铝壳定位夹爪气缸夹紧[A]
ANDLD
ANDNOT 501.05  ; RK_05 #1入壳铝壳定位夹爪气缸张开条件
ANDNOT 301.04  ; RK_05 #1入壳铝壳定位夹爪气缸夹紧[Pls]
ANDNOT 301.05  ; RK_05 #1入壳铝壳定位夹爪气缸张开[Pls]
ANDNOT 801.04  ; RK_05 #1入壳铝壳定位夹爪气缸夹紧位标志[0001.04]
OUT 601.04  ; RK_05 #1入壳铝壳定位夹爪气缸夹紧[A]
LD TR0
AND D1046.13  ; RK_05 #1入壳机构铝壳定位夹爪气缸张开1（步）
OUT 501.05  ; RK_05 #1入壳铝壳定位夹爪气缸张开条件
TIMX(550) 0121 D18  ; 自动运行条件延时时间, RK_05 #1入壳铝壳定位夹爪气缸张开延时[A]
LD TR0
LD 501.05  ; RK_05 #1入壳铝壳定位夹爪气缸张开条件
AND T0121  ; RK_05 #1入壳铝壳定位夹爪气缸张开延时[A]
OR 601.05  ; RK_05 #1入壳铝壳定位夹爪气缸张开[A]
ANDLD
ANDNOT 501.04  ; RK_05 #1入壳铝壳定位夹爪气缸夹紧条件
ANDNOT 301.05  ; RK_05 #1入壳铝壳定位夹爪气缸张开[Pls]
ANDNOT 301.04  ; RK_05 #1入壳铝壳定位夹爪气缸夹紧[Pls]
ANDNOT 801.05  ; RK_05 #1入壳铝壳定位夹爪气缸张开位标志[0001.05]
OUT 601.05  ; RK_05 #1入壳铝壳定位夹爪气缸张开[A]

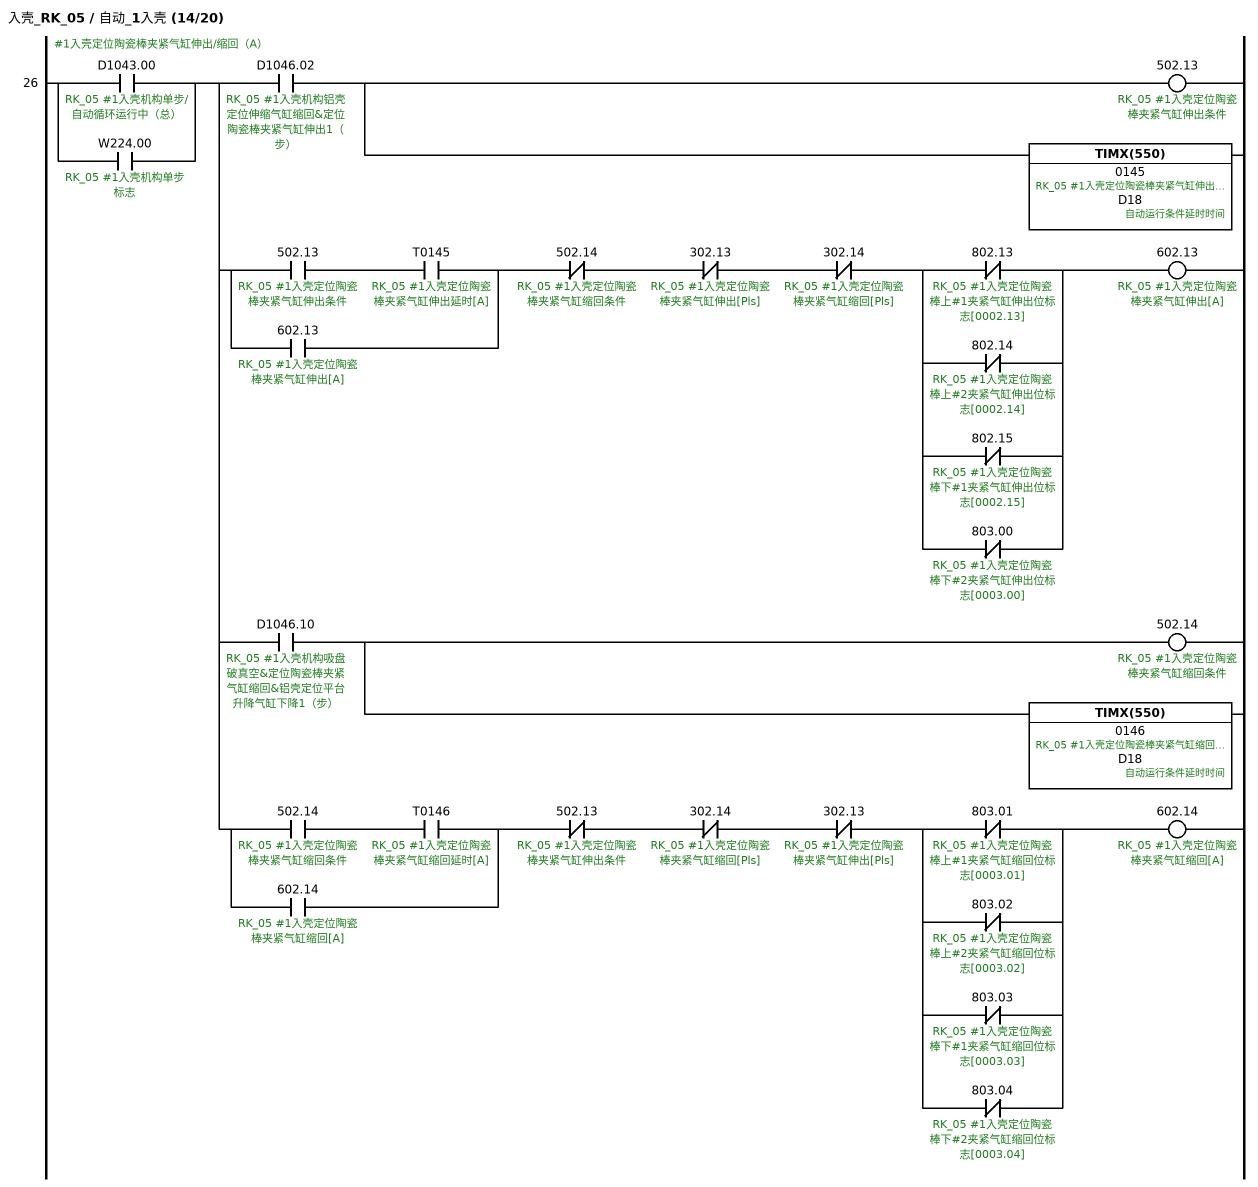
; rung 26: #1入壳定位陶瓷棒夹紧气缸伸出/缩回（A）
LD D1043.00  ; RK_05 #1入壳机构单步/自动循环运行中（总）
OR W224.00  ; RK_05 #1入壳机构单步标志
OUT TR0
AND D1046.02  ; RK_05 #1入壳机构铝壳定位伸缩气缸缩回&定位陶瓷棒夹紧气缸伸出1（步）
OUT 502.13  ; RK_05 #1入壳定位陶瓷棒夹紧气缸伸出条件
TIMX(550) 0145 D18  ; 自动运行条件延时时间, RK_05 #1入壳定位陶瓷棒夹紧气缸伸出延时[A]
LD TR0
LD 502.13  ; RK_05 #1入壳定位陶瓷棒夹紧气缸伸出条件
AND T0145  ; RK_05 #1入壳定位陶瓷棒夹紧气缸伸出延时[A]
OR 602.13  ; RK_05 #1入壳定位陶瓷棒夹紧气缸伸出[A]
ANDLD
ANDNOT 502.14  ; RK_05 #1入壳定位陶瓷棒夹紧气缸缩回条件
ANDNOT 302.13  ; RK_05 #1入壳定位陶瓷棒夹紧气缸伸出[Pls]
ANDNOT 302.14  ; RK_05 #1入壳定位陶瓷棒夹紧气缸缩回[Pls]
LDNOT 802.13  ; RK_05 #1入壳定位陶瓷棒上#1夹紧气缸伸出位标志[0002.13]
ORNOT 802.14  ; RK_05 #1入壳定位陶瓷棒上#2夹紧气缸伸出位标志[0002.14]
ORNOT 802.15  ; RK_05 #1入壳定位陶瓷棒下#1夹紧气缸伸出位标志[0002.15]
ORNOT 803.00  ; RK_05 #1入壳定位陶瓷棒下#2夹紧气缸伸出位标志[0003.00]
ANDLD
OUT 602.13  ; RK_05 #1入壳定位陶瓷棒夹紧气缸伸出[A]
LD TR0
AND D1046.10  ; RK_05 #1入壳机构吸盘破真空&定位陶瓷棒夹紧气缸缩回&铝壳定位平台升降气缸下降1（步）
OUT 502.14  ; RK_05 #1入壳定位陶瓷棒夹紧气缸缩回条件
TIMX(550) 0146 D18  ; 自动运行条件延时时间, RK_05 #1入壳定位陶瓷棒夹紧气缸缩回延时[A]
LD TR0
LD 502.14  ; RK_05 #1入壳定位陶瓷棒夹紧气缸缩回条件
AND T0146  ; RK_05 #1入壳定位陶瓷棒夹紧气缸缩回延时[A]
OR 602.14  ; RK_05 #1入壳定位陶瓷棒夹紧气缸缩回[A]
ANDLD
ANDNOT 502.13  ; RK_05 #1入壳定位陶瓷棒夹紧气缸伸出条件
ANDNOT 302.14  ; RK_05 #1入壳定位陶瓷棒夹紧气缸缩回[Pls]
ANDNOT 302.13  ; RK_05 #1入壳定位陶瓷棒夹紧气缸伸出[Pls]
LDNOT 803.01  ; RK_05 #1入壳定位陶瓷棒上#1夹紧气缸缩回位标志[0003.01]
ORNOT 803.02  ; RK_05 #1入壳定位陶瓷棒上#2夹紧气缸缩回位标志[0003.02]
ORNOT 803.03  ; RK_05 #1入壳定位陶瓷棒下#1夹紧气缸缩回位标志[0003.03]
ORNOT 803.04  ; RK_05 #1入壳定位陶瓷棒下#2夹紧气缸缩回位标志[0003.04]
ANDLD
OUT 602.14  ; RK_05 #1入壳定位陶瓷棒夹紧气缸缩回[A]

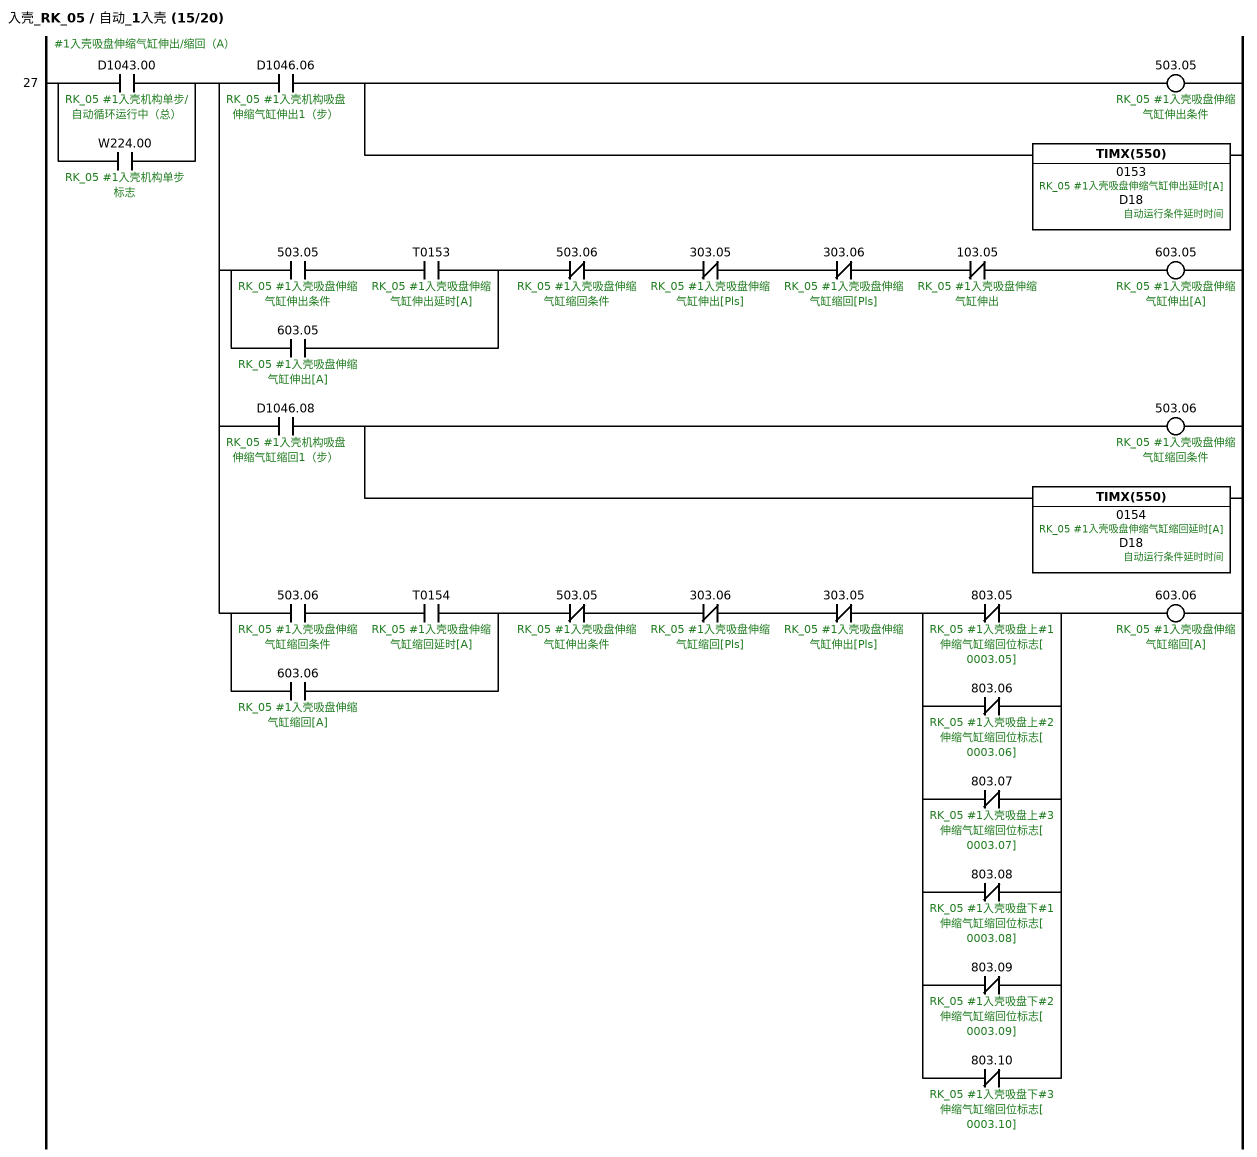
; rung 27: #1入壳吸盘伸缩气缸伸出/缩回（A）
LD D1043.00  ; RK_05 #1入壳机构单步/自动循环运行中（总）
OR W224.00  ; RK_05 #1入壳机构单步标志
OUT TR0
AND D1046.06  ; RK_05 #1入壳机构吸盘伸缩气缸伸出1（步）
OUT 503.05  ; RK_05 #1入壳吸盘伸缩气缸伸出条件
TIMX(550) 0153 D18  ; 自动运行条件延时时间, RK_05 #1入壳吸盘伸缩气缸伸出延时[A]
LD TR0
LD 503.05  ; RK_05 #1入壳吸盘伸缩气缸伸出条件
AND T0153  ; RK_05 #1入壳吸盘伸缩气缸伸出延时[A]
OR 603.05  ; RK_05 #1入壳吸盘伸缩气缸伸出[A]
ANDLD
ANDNOT 503.06  ; RK_05 #1入壳吸盘伸缩气缸缩回条件
ANDNOT 303.05  ; RK_05 #1入壳吸盘伸缩气缸伸出[Pls]
ANDNOT 303.06  ; RK_05 #1入壳吸盘伸缩气缸缩回[Pls]
ANDNOT 103.05  ; RK_05 #1入壳吸盘伸缩气缸伸出
OUT 603.05  ; RK_05 #1入壳吸盘伸缩气缸伸出[A]
LD TR0
AND D1046.08  ; RK_05 #1入壳机构吸盘伸缩气缸缩回1（步）
OUT 503.06  ; RK_05 #1入壳吸盘伸缩气缸缩回条件
TIMX(550) 0154 D18  ; 自动运行条件延时时间, RK_05 #1入壳吸盘伸缩气缸缩回延时[A]
LD TR0
LD 503.06  ; RK_05 #1入壳吸盘伸缩气缸缩回条件
AND T0154  ; RK_05 #1入壳吸盘伸缩气缸缩回延时[A]
OR 603.06  ; RK_05 #1入壳吸盘伸缩气缸缩回[A]
ANDLD
ANDNOT 503.05  ; RK_05 #1入壳吸盘伸缩气缸伸出条件
ANDNOT 303.06  ; RK_05 #1入壳吸盘伸缩气缸缩回[Pls]
ANDNOT 303.05  ; RK_05 #1入壳吸盘伸缩气缸伸出[Pls]
LDNOT 803.05  ; RK_05 #1入壳吸盘上#1伸缩气缸缩回位标志[0003.05]
ORNOT 803.06  ; RK_05 #1入壳吸盘上#2伸缩气缸缩回位标志[0003.06]
ORNOT 803.07  ; RK_05 #1入壳吸盘上#3伸缩气缸缩回位标志[0003.07]
ORNOT 803.08  ; RK_05 #1入壳吸盘下#1伸缩气缸缩回位标志[0003.08]
ORNOT 803.09  ; RK_05 #1入壳吸盘下#2伸缩气缸缩回位标志[0003.09]
ORNOT 803.10  ; RK_05 #1入壳吸盘下#3伸缩气缸缩回位标志[0003.10]
ANDLD
OUT 603.06  ; RK_05 #1入壳吸盘伸缩气缸缩回[A]

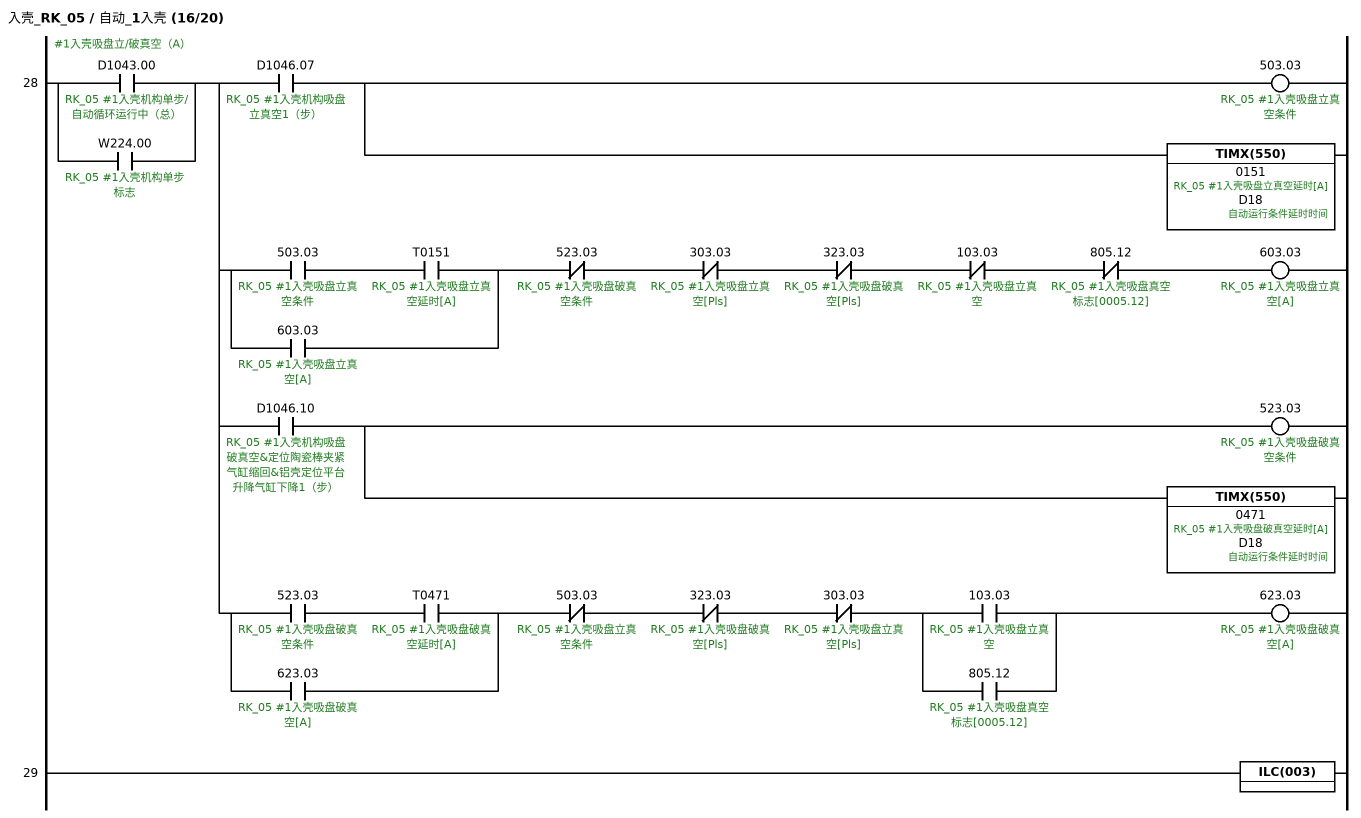
; rung 28: #1入壳吸盘立/破真空（A）
LD D1043.00  ; RK_05 #1入壳机构单步/自动循环运行中（总）
OR W224.00  ; RK_05 #1入壳机构单步标志
OUT TR0
AND D1046.07  ; RK_05 #1入壳机构吸盘立真空1（步）
OUT 503.03  ; RK_05 #1入壳吸盘立真空条件
TIMX(550) 0151 D18  ; 自动运行条件延时时间, RK_05 #1入壳吸盘立真空延时[A]
LD TR0
LD 503.03  ; RK_05 #1入壳吸盘立真空条件
AND T0151  ; RK_05 #1入壳吸盘立真空延时[A]
OR 603.03  ; RK_05 #1入壳吸盘立真空[A]
ANDLD
ANDNOT 523.03  ; RK_05 #1入壳吸盘破真空条件
ANDNOT 303.03  ; RK_05 #1入壳吸盘立真空[Pls]
ANDNOT 323.03  ; RK_05 #1入壳吸盘破真空[Pls]
ANDNOT 103.03  ; RK_05 #1入壳吸盘立真空
ANDNOT 805.12  ; RK_05 #1入壳吸盘真空标志[0005.12]
OUT 603.03  ; RK_05 #1入壳吸盘立真空[A]
LD TR0
AND D1046.10  ; RK_05 #1入壳机构吸盘破真空&定位陶瓷棒夹紧气缸缩回&铝壳定位平台升降气缸下降1（步）
OUT 523.03  ; RK_05 #1入壳吸盘破真空条件
TIMX(550) 0471 D18  ; 自动运行条件延时时间, RK_05 #1入壳吸盘破真空延时[A]
LD TR0
LD 523.03  ; RK_05 #1入壳吸盘破真空条件
AND T0471  ; RK_05 #1入壳吸盘破真空延时[A]
OR 623.03  ; RK_05 #1入壳吸盘破真空[A]
ANDLD
ANDNOT 503.03  ; RK_05 #1入壳吸盘立真空条件
ANDNOT 323.03  ; RK_05 #1入壳吸盘破真空[Pls]
ANDNOT 303.03  ; RK_05 #1入壳吸盘立真空[Pls]
LD 103.03  ; RK_05 #1入壳吸盘立真空
OR 805.12  ; RK_05 #1入壳吸盘真空标志[0005.12]
ANDLD
OUT 623.03  ; RK_05 #1入壳吸盘破真空[A]
; rung 29
ILC(003)

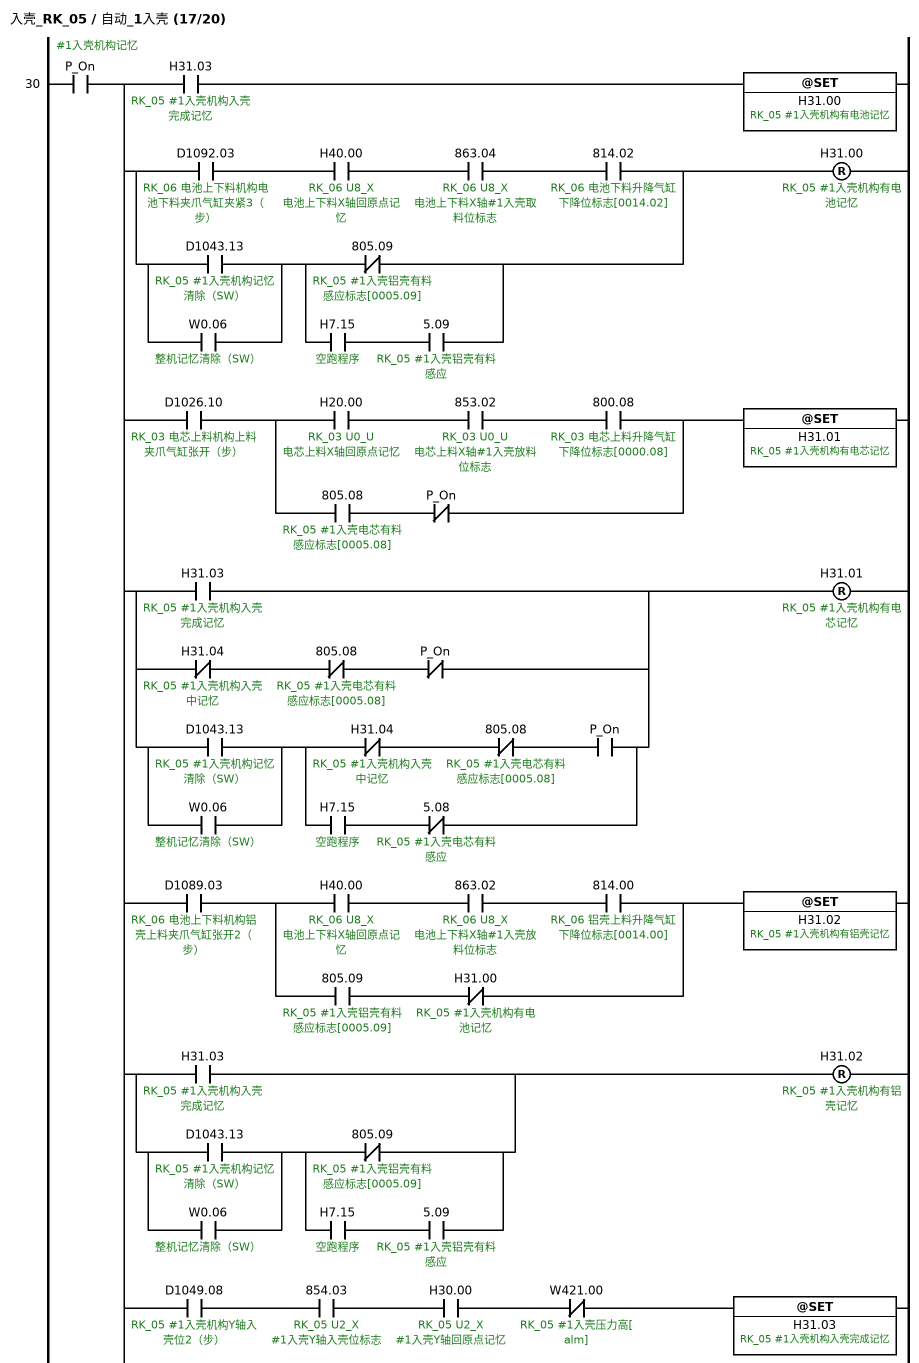

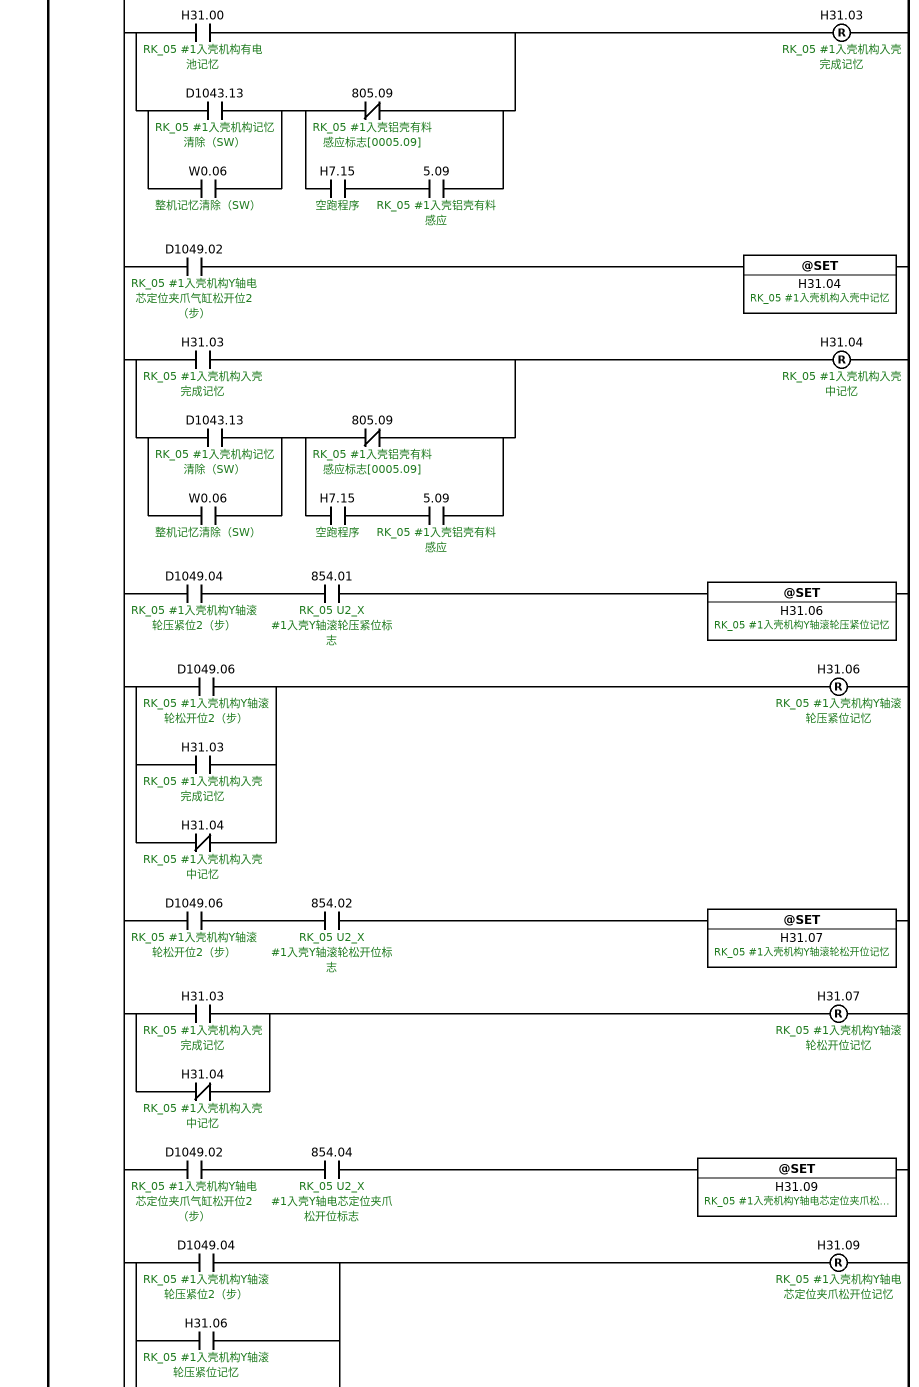

